   REGION Output Mapping
       // TwoWayActuator
       "Unit1.Em0.HmiInterface".cmStacker1NgBoxClampMoverOpenClose.commands := "ManualOperationControl_U1Em0".twoWayActuator[1].commands;
       "Unit1.Em0.HmiInterface".cmStacker1NgBoxClampLeftOpenClose.commands := "ManualOperationControl_U1Em0".twoWayActuator[2].commands;
       "Unit1.Em0.HmiInterface".cmStacker1NgBoxClampRightOpenClose.commands := "ManualOperationControl_U1Em0".twoWayActuator[3].commands;
       "Unit1.Em0.HmiInterface".cmStacker1NgBoxLoadingUpDown.commands := "ManualOperationControl_U1Em0".twoWayActuator[4].commands;
       "Unit1.Em0.HmiInterface".cmStacker1NgBoxUnitMoverBwdFwd.commands := "ManualOperationControl_U1Em0".twoWayActuator[5].commands;
       "Unit1.Em0.HmiInterface".cmStacker1NgBoxLiftDownUp.commands := "ManualOperationControl_U1Em0".twoWayActuator[6].commands;
       "Unit1.Em0.HmiInterface".cmStacker1NgBoxLockDownUp.commands := "ManualOperationControl_U1Em0".twoWayActuator[7].commands;
   END_REGION
END_REGION

REGION Network 3: Equipment Module 0
   RUNG wire#powerrail
      "CallManualOperationLines_EM"(disableUnit := #disableUnit1, manualOperationEm := "ManualOperationControl_U1Em0".manualOperationEm, manualOperationEmArea := "ManualOperationControl_U1Em0".manualOperationEmArea, manualOperationCms := "ManualOperationControl_U1Em0".manualOperationCms, Axis64Pos := "ManualOperationControl_U1Em0".axis, AxisSoftCam := "ManualOperationControl_U1Em0".softCam, twoWayAcutor := "ManualOperationControl_U1Em0".twoWayActuator, Status := #StatusEm[0].Status, errorID := #errorIDEm[0].errorID)
   END_RUNG
   // the same network as SCL:
   "CallManualOperationLines_EM"(disableUnit := #disableUnit1,
                           manualOperationEm := "ManualOperationControl_U1Em0".manualOperationEm,
                           manualOperationEmArea := "ManualOperationControl_U1Em0".manualOperationEmArea,
                           manualOperationCms := "ManualOperationControl_U1Em0".manualOperationCms,
                           Axis64Pos := "ManualOperationControl_U1Em0".axis,
                           AxisSoftCam := "ManualOperationControl_U1Em0".softCam,
                           twoWayAcutor := "ManualOperationControl_U1Em0".twoWayActuator,
                           Status := #StatusEm[0].Status,
                           errorID := #errorIDEm[0].errorID);
END_REGION

REGION Network 4 (SCL): Equipment Module 1 Cms Mapping
   REGION Input Mapping
       // TwoWayActuator
       "ManualOperationControl_U1Em1".twoWayActuator[1].monitoring := "Unit1.Em1.HmiInterface".cmStacker2NgBoxClampMoverOpenClose.monitoring;
       "ManualOperationControl_U1Em1".twoWayActuator[2].monitoring := "Unit1.Em1.HmiInterface".cmStacker2NgBoxClampLeftOpenClose.monitoring;
       "ManualOperationControl_U1Em1".twoWayActuator[3].monitoring := "Unit1.Em1.HmiInterface".cmStacker2NgBoxClampRightOpenClose.monitoring;
       "ManualOperationControl_U1Em1".twoWayActuator[4].monitoring := "Unit1.Em1.HmiInterface".cmStacker2NgBoxLoadingUpDown.monitoring;
       "ManualOperationControl_U1Em1".twoWayActuator[5].monitoring := "Unit1.Em1.HmiInterface".cmStacker2NgBoxUnitMoverBwdFwd.monitoring;
       "ManualOperationControl_U1Em1".twoWayActuator[6].monitoring := "Unit1.Em1.HmiInterface".cmStacker2NgBoxLiftDownUp.monitoring;
       "ManualOperationControl_U1Em1".twoWayActuator[7].monitoring := "Unit1.Em1.HmiInterface".cmStacker2NgBoxLockDownUp.monitoring;
   END_REGION


   REGION Output Mapping  
       // TwoWayActuator
       "Unit1.Em1.HmiInterface".cmStacker2NgBoxClampMoverOpenClose.commands := "ManualOperationControl_U1Em1".twoWayActuator[1].commands;
       "Unit1.Em1.HmiInterface".cmStacker2NgBoxClampLeftOpenClose.commands := "ManualOperationControl_U1Em1".twoWayActuator[2].commands;
       "Unit1.Em1.HmiInterface".cmStacker2NgBoxClampRightOpenClose.commands := "ManualOperationControl_U1Em1".twoWayActuator[3].commands;
       "Unit1.Em1.HmiInterface".cmStacker2NgBoxLoadingUpDown.commands := "ManualOperationControl_U1Em1".twoWayActuator[4].commands;
       "Unit1.Em1.HmiInterface".cmStacker2NgBoxUnitMoverBwdFwd.commands := "ManualOperationControl_U1Em1".twoWayActuator[5].commands;
       "Unit1.Em1.HmiInterface".cmStacker2NgBoxLiftDownUp.commands := "ManualOperationControl_U1Em1".twoWayActuator[6].commands;
       "Unit1.Em1.HmiInterface".cmStacker2NgBoxLockDownUp.commands := "ManualOperationControl_U1Em1".twoWayActuator[7].commands;
   END_REGION
END_REGION

REGION Network 5: Equipment Module 1
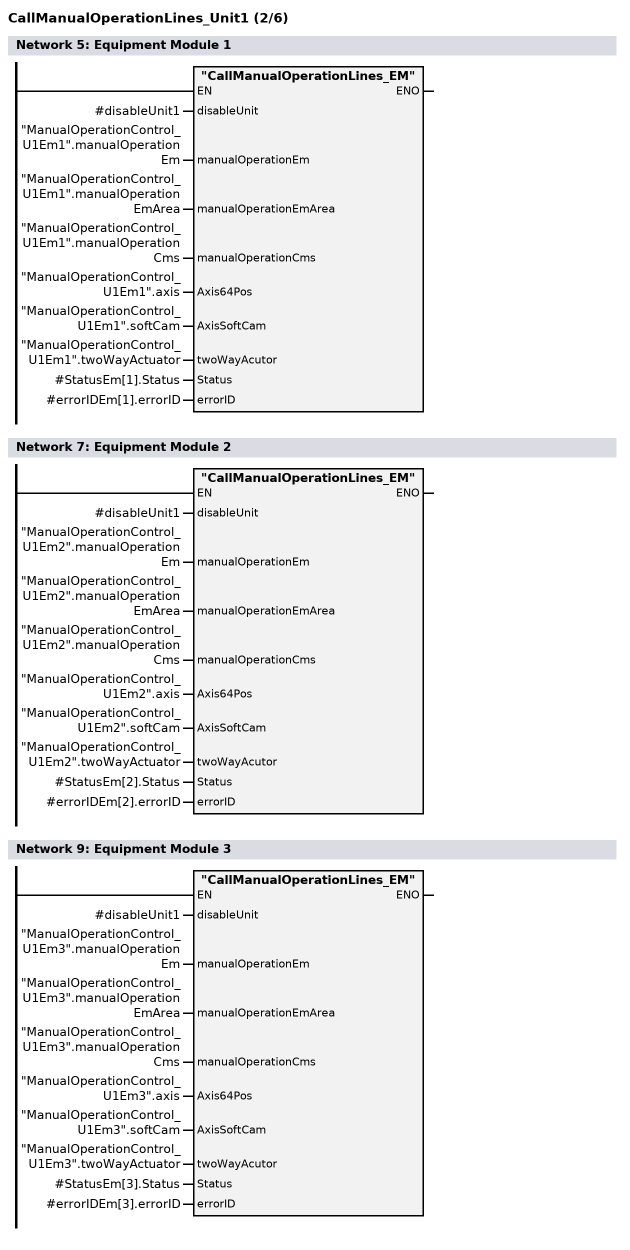
   RUNG wire#powerrail
      "CallManualOperationLines_EM"(disableUnit := #disableUnit1, manualOperationEm := "ManualOperationControl_U1Em1".manualOperationEm, manualOperationEmArea := "ManualOperationControl_U1Em1".manualOperationEmArea, manualOperationCms := "ManualOperationControl_U1Em1".manualOperationCms, Axis64Pos := "ManualOperationControl_U1Em1".axis, AxisSoftCam := "ManualOperationControl_U1Em1".softCam, twoWayAcutor := "ManualOperationControl_U1Em1".twoWayActuator, Status := #StatusEm[1].Status, errorID := #errorIDEm[1].errorID)
   END_RUNG
   // the same network as SCL:
   "CallManualOperationLines_EM"(disableUnit := #disableUnit1,
                           manualOperationEm := "ManualOperationControl_U1Em1".manualOperationEm,
                           manualOperationEmArea := "ManualOperationControl_U1Em1".manualOperationEmArea,
                           manualOperationCms := "ManualOperationControl_U1Em1".manualOperationCms,
                           Axis64Pos := "ManualOperationControl_U1Em1".axis,
                           AxisSoftCam := "ManualOperationControl_U1Em1".softCam,
                           twoWayAcutor := "ManualOperationControl_U1Em1".twoWayActuator,
                           Status := #StatusEm[1].Status,
                           errorID := #errorIDEm[1].errorID);
END_REGION

REGION Network 6 (SCL): Equipment Module 2 Cms Mapping
   REGION Input Mapping
       // Axis
       "ManualOperationControl_U1Em2".axis[1].monitoring := "Unit1.Em2.HmiInterface".cmJROutPnPLeftAxisX.monitoring;
       "ManualOperationControl_U1Em2".axis[2].monitoring := "Unit1.Em2.HmiInterface".cmJROutPnPLeftAxisZ.monitoring;
       "ManualOperationControl_U1Em2".axis[3].monitoring := "Unit1.Em2.HmiInterface".cmJROutPnPRightAxisX.monitoring;
       "ManualOperationControl_U1Em2".axis[4].monitoring := "Unit1.Em2.HmiInterface".cmJROutPnPRightAxisZ.monitoring;

       // SoftCam
       "ManualOperationControl_U1Em2".softCam[1] := "Unit1.Em2.HmiInterface".cm.softcam.jrOutPnPLeftAxisX;
       "ManualOperationControl_U1Em2".softCam[2] := "Unit1.Em2.HmiInterface".cm.softcam.jrOutPnPLeftAxisZ;
       "ManualOperationControl_U1Em2".softCam[3] := "Unit1.Em2.HmiInterface".cm.softcam.jrOutPnPRightAxisX;
       "ManualOperationControl_U1Em2".softCam[4] := "Unit1.Em2.HmiInterface".cm.softcam.jrOutPnPRightAxisZ;

       // TwoWayActuator
       "ManualOperationControl_U1Em2".twoWayActuator[1].monitoring := "Unit1.Em2.HmiInterface".cmJROutPnPLeftClampOpenClose.monitoring;
       "ManualOperationControl_U1Em2".twoWayActuator[2].monitoring := "Unit1.Em2.HmiInterface".cmJROutPnPRightClampOpenClose.monitoring;
   END_REGION


   REGION Output Mapping
       // Axis
       "Unit1.Em2.HmiInterface".cmJROutPnPLeftAxisX.commands.jogForward := "ManualOperationControl_U1Em2".axis[1].commands.jogForward;
       "Unit1.Em2.HmiInterface".cmJROutPnPLeftAxisX.commands.jogBackward := "ManualOperationControl_U1Em2".axis[1].commands.jogBackward;
       "Unit1.Em2.HmiInterface".cmJROutPnPLeftAxisZ.commands.jogForward := "ManualOperationControl_U1Em2".axis[2].commands.jogForward;
       "Unit1.Em2.HmiInterface".cmJROutPnPLeftAxisZ.commands.jogBackward := "ManualOperationControl_U1Em2".axis[2].commands.jogBackward;
       "Unit1.Em2.HmiInterface".cmJROutPnPRightAxisX.commands.jogForward := "ManualOperationControl_U1Em2".axis[3].commands.jogForward;
       "Unit1.Em2.HmiInterface".cmJROutPnPRightAxisX.commands.jogBackward := "ManualOperationControl_U1Em2".axis[3].commands.jogBackward;
       "Unit1.Em2.HmiInterface".cmJROutPnPRightAxisZ.commands.jogForward := "ManualOperationControl_U1Em2".axis[4].commands.jogForward;
       "Unit1.Em2.HmiInterface".cmJROutPnPRightAxisZ.commands.jogBackward := "ManualOperationControl_U1Em2".axis[4].commands.jogBackward;

       // TwoWayActuator
       "Unit1.Em2.HmiInterface".cmJROutPnPLeftClampOpenClose.commands := "ManualOperationControl_U1Em2".twoWayActuator[1].commands;
       "Unit1.Em2.HmiInterface".cmJROutPnPRightClampOpenClose.commands := "ManualOperationControl_U1Em2".twoWayActuator[2].commands;
   END_REGION
END_REGION

REGION Network 7: Equipment Module 2
   RUNG wire#powerrail
      "CallManualOperationLines_EM"(disableUnit := #disableUnit1, manualOperationEm := "ManualOperationControl_U1Em2".manualOperationEm, manualOperationEmArea := "ManualOperationControl_U1Em2".manualOperationEmArea, manualOperationCms := "ManualOperationControl_U1Em2".manualOperationCms, Axis64Pos := "ManualOperationControl_U1Em2".axis, AxisSoftCam := "ManualOperationControl_U1Em2".softCam, twoWayAcutor := "ManualOperationControl_U1Em2".twoWayActuator, Status := #StatusEm[2].Status, errorID := #errorIDEm[2].errorID)
   END_RUNG
   // the same network as SCL:
   "CallManualOperationLines_EM"(disableUnit := #disableUnit1,
                           manualOperationEm := "ManualOperationControl_U1Em2".manualOperationEm,
                           manualOperationEmArea := "ManualOperationControl_U1Em2".manualOperationEmArea,
                           manualOperationCms := "ManualOperationControl_U1Em2".manualOperationCms,
                           Axis64Pos := "ManualOperationControl_U1Em2".axis,
                           AxisSoftCam := "ManualOperationControl_U1Em2".softCam,
                           twoWayAcutor := "ManualOperationControl_U1Em2".twoWayActuator,
                           Status := #StatusEm[2].Status,
                           errorID := #errorIDEm[2].errorID);
END_REGION

REGION Network 8 (SCL): Equipment Module 3 Cms Mapping
   REGION Input Mapping
        // Axis
       "ManualOperationControl_U1Em3".axis[1].monitoring := "Unit1.Em3.HmiInterface".cmTopTapeAxisX.monitoring;
       "ManualOperationControl_U1Em3".axis[2].monitoring := "Unit1.Em3.HmiInterface".cmTopTapeAxisY.monitoring;

       // SoftCam
       "ManualOperationControl_U1Em3".softCam[1] := "Unit1.Em3.HmiInterface".cm.softcam.topTapeAxisX;
       "ManualOperationControl_U1Em3".softCam[2] := "Unit1.Em3.HmiInterface".cm.softcam.topTapeAxisY;

       // TwoWayActuator
       "ManualOperationControl_U1Em3".twoWayActuator[1].monitoring := "Unit1.Em3.HmiInterface".cmTopTapeCutterUpDown.monitoring;
       "ManualOperationControl_U1Em3".twoWayActuator[2].monitoring := "Unit1.Em3.HmiInterface".cmTopTapeCutterClampUpDown.monitoring;
       "ManualOperationControl_U1Em3".twoWayActuator[3].monitoring := "Unit1.Em3.HmiInterface".cmTopTapeLoadingClampOpenClose.monitoring;
       "ManualOperationControl_U1Em3".twoWayActuator[4].monitoring := "Unit1.Em3.HmiInterface".cmTopTapeTensionBwdFwd.monitoring;
       "ManualOperationControl_U1Em3".twoWayActuator[5].monitoring := "Unit1.Em3.HmiInterface".cmTopTapeLoadingBwdFwd.monitoring;
       "ManualOperationControl_U1Em3".twoWayActuator[6].monitoring := "Unit1.Em3.HmiInterface".cmTopTapeClampTopLeftUpDown.monitoring;
       "ManualOperationControl_U1Em3".twoWayActuator[7].monitoring := "Unit1.Em3.HmiInterface".cmTopTapeClampTopCenterUpDown.monitoring;
       "ManualOperationControl_U1Em3".twoWayActuator[8].monitoring := "Unit1.Em3.HmiInterface".cmTopTapeClampTopRightUpDown.monitoring;
       "ManualOperationControl_U1Em3".twoWayActuator[9].monitoring := "Unit1.Em3.HmiInterface".cmTopTapeClampBtmDownUp.monitoring;
       "ManualOperationControl_U1Em3".twoWayActuator[10].monitoring := "Unit1.Em3.HmiInterface".cmTopTapeAttachmentUpDown.monitoring;
       "ManualOperationControl_U1Em3".twoWayActuator[11].monitoring := "Unit1.Em3.HmiInterface".cmTopTapeAttachmentVaccumOffOn.monitoring;

   END_REGION


   REGION Output Mapping
       // Axis
       "Unit1.Em3.HmiInterface".cmTopTapeAxisX.commands.jogForward := "ManualOperationControl_U1Em3".axis[1].commands.jogForward;
       "Unit1.Em3.HmiInterface".cmTopTapeAxisX.commands.jogBackward := "ManualOperationControl_U1Em3".axis[1].commands.jogBackward;
       "Unit1.Em3.HmiInterface".cmTopTapeAxisY.commands.jogForward := "ManualOperationControl_U1Em3".axis[2].commands.jogForward;
       "Unit1.Em3.HmiInterface".cmTopTapeAxisY.commands.jogBackward := "ManualOperationControl_U1Em3".axis[2].commands.jogBackward;

       // TwoWayActuator
       "Unit1.Em3.HmiInterface".cmTopTapeCutterUpDown.commands := "ManualOperationControl_U1Em3".twoWayActuator[1].commands;
       "Unit1.Em3.HmiInterface".cmTopTapeCutterClampUpDown.commands := "ManualOperationControl_U1Em3".twoWayActuator[2].commands;
       "Unit1.Em3.HmiInterface".cmTopTapeLoadingClampOpenClose.commands := "ManualOperationControl_U1Em3".twoWayActuator[3].commands;
       "Unit1.Em3.HmiInterface".cmTopTapeTensionBwdFwd.commands := "ManualOperationControl_U1Em3".twoWayActuator[4].commands;
       "Unit1.Em3.HmiInterface".cmTopTapeLoadingBwdFwd.commands := "ManualOperationControl_U1Em3".twoWayActuator[5].commands;
       "Unit1.Em3.HmiInterface".cmTopTapeClampTopLeftUpDown.commands := "ManualOperationControl_U1Em3".twoWayActuator[6].commands;
       "Unit1.Em3.HmiInterface".cmTopTapeClampTopCenterUpDown.commands := "ManualOperationControl_U1Em3".twoWayActuator[7].commands;
       "Unit1.Em3.HmiInterface".cmTopTapeClampTopRightUpDown.commands := "ManualOperationControl_U1Em3".twoWayActuator[8].commands;
       "Unit1.Em3.HmiInterface".cmTopTapeClampBtmDownUp.commands := "ManualOperationControl_U1Em3".twoWayActuator[9].commands;
       "Unit1.Em3.HmiInterface".cmTopTapeAttachmentUpDown.commands := "ManualOperationControl_U1Em3".twoWayActuator[10].commands;
       "Unit1.Em3.HmiInterface".cmTopTapeAttachmentVaccumOffOn.commands := "ManualOperationControl_U1Em3".twoWayActuator[11].commands;

   END_REGION
END_REGION

REGION Network 9: Equipment Module 3
   RUNG wire#powerrail
      "CallManualOperationLines_EM"(disableUnit := #disableUnit1, manualOperationEm := "ManualOperationControl_U1Em3".manualOperationEm, manualOperationEmArea := "ManualOperationControl_U1Em3".manualOperationEmArea, manualOperationCms := "ManualOperationControl_U1Em3".manualOperationCms, Axis64Pos := "ManualOperationControl_U1Em3".axis, AxisSoftCam := "ManualOperationControl_U1Em3".softCam, twoWayAcutor := "ManualOperationControl_U1Em3".twoWayActuator, Status := #StatusEm[3].Status, errorID := #errorIDEm[3].errorID)
   END_RUNG
   // the same network as SCL:
   "CallManualOperationLines_EM"(disableUnit := #disableUnit1,
                           manualOperationEm := "ManualOperationControl_U1Em3".manualOperationEm,
                           manualOperationEmArea := "ManualOperationControl_U1Em3".manualOperationEmArea,
                           manualOperationCms := "ManualOperationControl_U1Em3".manualOperationCms,
                           Axis64Pos := "ManualOperationControl_U1Em3".axis,
                           AxisSoftCam := "ManualOperationControl_U1Em3".softCam,
                           twoWayAcutor := "ManualOperationControl_U1Em3".twoWayActuator,
                           Status := #StatusEm[3].Status,
                           errorID := #errorIDEm[3].errorID);
END_REGION

REGION Network 10 (SCL): Equipment Module 4 Cms Mapping
   REGION Input Mapping
       // Axis
       "ManualOperationControl_U1Em4".axis[1].monitoring := "Unit1.Em4.HmiInterface".cmSideTapeFixStageAxisX.monitoring;
       "ManualOperationControl_U1Em4".axis[2].monitoring := "Unit1.Em4.HmiInterface".cmSideTapeFixStageAxisC.monitoring;
       "ManualOperationControl_U1Em4".axis[3].monitoring := "Unit1.Em4.HmiInterface".cmSideTapeAttachmentAxisX.monitoring;
       "ManualOperationControl_U1Em4".axis[4].monitoring := "Unit1.Em4.HmiInterface".cmSideTapeAttachmentAxisY.monitoring;

       // SoftCam
       "ManualOperationControl_U1Em4".softCam[1] := "Unit1.Em4.HmiInterface".cm.softcam.sideTapeFixStageAxisX;
       "ManualOperationControl_U1Em4".softCam[2] := "Unit1.Em4.HmiInterface".cm.softcam.sideTapeFixStageAxisC;
       "ManualOperationControl_U1Em4".softCam[3] := "Unit1.Em4.HmiInterface".cm.softcam.sideTapeAttachmentAxisX;
       "ManualOperationControl_U1Em4".softCam[4] := "Unit1.Em4.HmiInterface".cm.softcam.sideTapeAttachmentAxisY;

       // TwoWayActuator
       "ManualOperationControl_U1Em4".twoWayActuator[1].monitoring := "Unit1.Em4.HmiInterface".cmSideTapeCutterBwdFwd.monitoring;
       "ManualOperationControl_U1Em4".twoWayActuator[2].monitoring := "Unit1.Em4.HmiInterface".cmSideTapeCutterClampBwdFwd.monitoring;
       "ManualOperationControl_U1Em4".twoWayActuator[3].monitoring := "Unit1.Em4.HmiInterface".cmSideTapeLoadingClampOpenClose.monitoring;
       "ManualOperationControl_U1Em4".twoWayActuator[4].monitoring := "Unit1.Em4.HmiInterface".cmSideTapeLoadingDownUp.monitoring;
       "ManualOperationControl_U1Em4".twoWayActuator[5].monitoring := "Unit1.Em4.HmiInterface".cmSideTapeTensionBwdFwd.monitoring;
       "ManualOperationControl_U1Em4".twoWayActuator[6].monitoring := "Unit1.Em4.HmiInterface".cmSideTapeAttachmentLeftBwdFwd.monitoring;
       "ManualOperationControl_U1Em4".twoWayActuator[7].monitoring := "Unit1.Em4.HmiInterface".cmSideTapeAttachmentRightBwdFwd.monitoring;
       "ManualOperationControl_U1Em4".twoWayActuator[8].monitoring := "Unit1.Em4.HmiInterface".cmSideTapeAttachmentBtmBwdFwd.monitoring;
       "ManualOperationControl_U1Em4".twoWayActuator[9].monitoring := "Unit1.Em4.HmiInterface".cmSideTapeFixStageClampOpenClose.monitoring;
       "ManualOperationControl_U1Em4".twoWayActuator[10].monitoring := "Unit1.Em4.HmiInterface".cmSideTapeAttachment1TopVaccumOffOn.monitoring;
       "ManualOperationControl_U1Em4".twoWayActuator[11].monitoring := "Unit1.Em4.HmiInterface".cmSideTapeAttachment1BtmVaccumOffOn.monitoring;
       "ManualOperationControl_U1Em4".twoWayActuator[12].monitoring := "Unit1.Em4.HmiInterface".cmSideTapeAttachment2TopVaccumOffOn.monitoring;
       "ManualOperationControl_U1Em4".twoWayActuator[13].monitoring := "Unit1.Em4.HmiInterface".cmSideTapeAttachment2BtmVaccumOffOn.monitoring;

   END_REGION


   REGION Output Mapping
       // Axis
       "Unit1.Em4.HmiInterface".cmSideTapeFixStageAxisX.commands.jogForward := "ManualOperationControl_U1Em4".axis[1].commands.jogForward;
       "Unit1.Em4.HmiInterface".cmSideTapeFixStageAxisX.commands.jogBackward := "ManualOperationControl_U1Em4".axis[1].commands.jogBackward;
       "Unit1.Em4.HmiInterface".cmSideTapeFixStageAxisC.commands.jogForward := "ManualOperationControl_U1Em4".axis[2].commands.jogForward;
       "Unit1.Em4.HmiInterface".cmSideTapeFixStageAxisC.commands.jogBackward := "ManualOperationControl_U1Em4".axis[2].commands.jogBackward;
       "Unit1.Em4.HmiInterface".cmSideTapeAttachmentAxisX.commands.jogForward := "ManualOperationControl_U1Em4".axis[3].commands.jogForward;
       "Unit1.Em4.HmiInterface".cmSideTapeAttachmentAxisX.commands.jogBackward := "ManualOperationControl_U1Em4".axis[3].commands.jogBackward;
       "Unit1.Em4.HmiInterface".cmSideTapeAttachmentAxisY.commands.jogForward := "ManualOperationControl_U1Em4".axis[4].commands.jogForward;
       "Unit1.Em4.HmiInterface".cmSideTapeAttachmentAxisY.commands.jogBackward := "ManualOperationControl_U1Em4".axis[4].commands.jogBackward;

       // TwoWayActuator
       "Unit1.Em4.HmiInterface".cmSideTapeCutterBwdFwd.commands := "ManualOperationControl_U1Em4".twoWayActuator[1].commands;
       "Unit1.Em4.HmiInterface".cmSideTapeCutterClampBwdFwd.commands := "ManualOperationControl_U1Em4".twoWayActuator[2].commands;
       "Unit1.Em4.HmiInterface".cmSideTapeLoadingClampOpenClose.commands := "ManualOperationControl_U1Em4".twoWayActuator[3].commands;
       "Unit1.Em4.HmiInterface".cmSideTapeLoadingDownUp.commands:= "ManualOperationControl_U1Em4".twoWayActuator[4].commands;
       "Unit1.Em4.HmiInterface".cmSideTapeTensionBwdFwd.commands := "ManualOperationControl_U1Em4".twoWayActuator[5].commands;
       "Unit1.Em4.HmiInterface".cmSideTapeAttachmentLeftBwdFwd.commands := "ManualOperationControl_U1Em4".twoWayActuator[6].commands;
       "Unit1.Em4.HmiInterface".cmSideTapeAttachmentRightBwdFwd.commands := "ManualOperationControl_U1Em4".twoWayActuator[7].commands;
       "Unit1.Em4.HmiInterface".cmSideTapeAttachmentBtmBwdFwd.commands := "ManualOperationControl_U1Em4".twoWayActuator[8].commands;
       "Unit1.Em4.HmiInterface".cmSideTapeFixStageClampOpenClose.commands := "ManualOperationControl_U1Em4".twoWayActuator[9].commands;
       "Unit1.Em4.HmiInterface".cmSideTapeAttachment1TopVaccumOffOn.commands := "ManualOperationControl_U1Em4".twoWayActuator[10].commands;
       "Unit1.Em4.HmiInterface".cmSideTapeAttachment1BtmVaccumOffOn.commands := "ManualOperationControl_U1Em4".twoWayActuator[11].commands;
       "Unit1.Em4.HmiInterface".cmSideTapeAttachment2TopVaccumOffOn.commands := "ManualOperationControl_U1Em4".twoWayActuator[12].commands;
       "Unit1.Em4.HmiInterface".cmSideTapeAttachment2BtmVaccumOffOn.commands := "ManualOperationControl_U1Em4".twoWayActuator[13].commands;

   END_REGION
END_REGION

REGION Network 11: Equipment Module 4
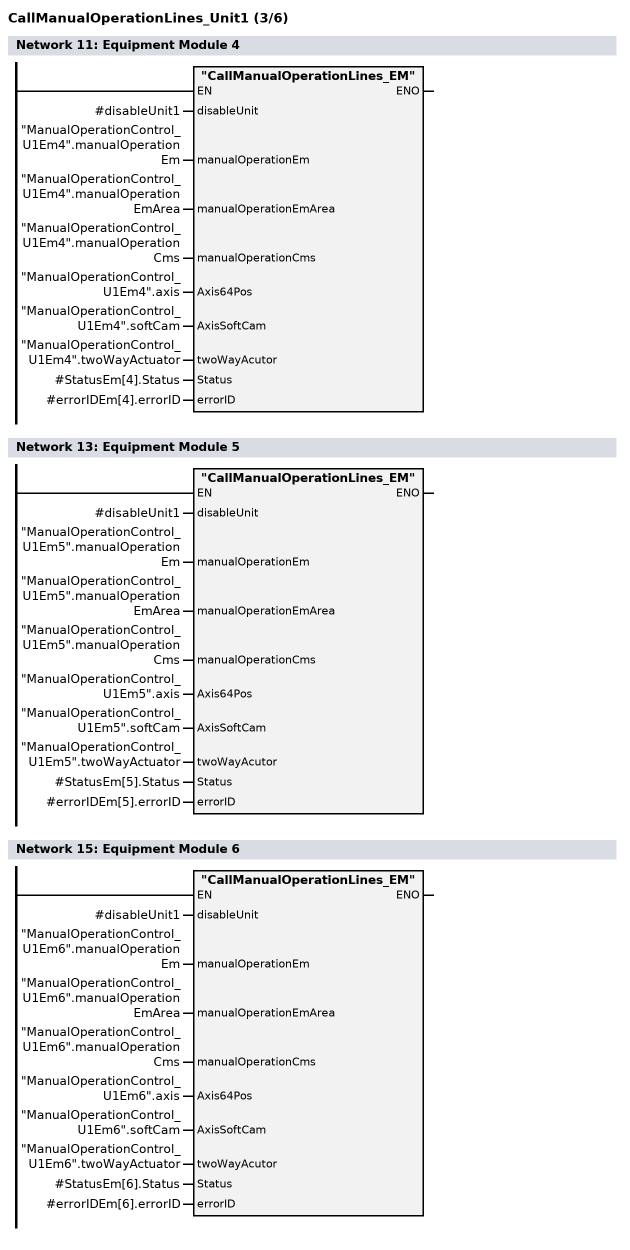
   RUNG wire#powerrail
      "CallManualOperationLines_EM"(disableUnit := #disableUnit1, manualOperationEm := "ManualOperationControl_U1Em4".manualOperationEm, manualOperationEmArea := "ManualOperationControl_U1Em4".manualOperationEmArea, manualOperationCms := "ManualOperationControl_U1Em4".manualOperationCms, Axis64Pos := "ManualOperationControl_U1Em4".axis, AxisSoftCam := "ManualOperationControl_U1Em4".softCam, twoWayAcutor := "ManualOperationControl_U1Em4".twoWayActuator, Status := #StatusEm[4].Status, errorID := #errorIDEm[4].errorID)
   END_RUNG
   // the same network as SCL:
   "CallManualOperationLines_EM"(disableUnit := #disableUnit1,
                           manualOperationEm := "ManualOperationControl_U1Em4".manualOperationEm,
                           manualOperationEmArea := "ManualOperationControl_U1Em4".manualOperationEmArea,
                           manualOperationCms := "ManualOperationControl_U1Em4".manualOperationCms,
                           Axis64Pos := "ManualOperationControl_U1Em4".axis,
                           AxisSoftCam := "ManualOperationControl_U1Em4".softCam,
                           twoWayAcutor := "ManualOperationControl_U1Em4".twoWayActuator,
                           Status := #StatusEm[4].Status,
                           errorID := #errorIDEm[4].errorID);
END_REGION

REGION Network 12 (SCL): Equipment Module 5 Cms Mapping
   REGION Input Mapping
        // Axis
       "ManualOperationControl_U1Em5".axis[1].monitoring := "Unit1.Em5.HmiInterface".cmTransferPnPLeftAxisX.monitoring;
       "ManualOperationControl_U1Em5".axis[2].monitoring := "Unit1.Em5.HmiInterface".cmTransferPnPLeftAxisY.monitoring;
       "ManualOperationControl_U1Em5".axis[3].monitoring := "Unit1.Em5.HmiInterface".cmTransferPnPLeftAxisZ.monitoring;
       "ManualOperationControl_U1Em5".axis[4].monitoring := "Unit1.Em5.HmiInterface".cmTransferPnPRightAxisX.monitoring;
       "ManualOperationControl_U1Em5".axis[5].monitoring := "Unit1.Em5.HmiInterface".cmTransferPnPRightAxisY.monitoring;
       "ManualOperationControl_U1Em5".axis[6].monitoring := "Unit1.Em5.HmiInterface".cmTransferPnPRightAxisZ.monitoring;

       // SoftCam
       "ManualOperationControl_U1Em5".softCam[1] := "Unit1.Em5.HmiInterface".cm.softcam.transferPnPLeftAxisX;
       "ManualOperationControl_U1Em5".softCam[2] := "Unit1.Em5.HmiInterface".cm.softcam.transferPnPLeftAxisY;
       "ManualOperationControl_U1Em5".softCam[3] := "Unit1.Em5.HmiInterface".cm.softcam.transferPnPLeftAxisZ;
       "ManualOperationControl_U1Em5".softCam[4] := "Unit1.Em5.HmiInterface".cm.softcam.transferPnPRightAxisX;
       "ManualOperationControl_U1Em5".softCam[5] := "Unit1.Em5.HmiInterface".cm.softcam.transferPnPRightAxisY;
       "ManualOperationControl_U1Em5".softCam[6] := "Unit1.Em5.HmiInterface".cm.softcam.transferPnPRightAxisZ;

       // TwoWayActuator
       "ManualOperationControl_U1Em5".twoWayActuator[1].monitoring := "Unit1.Em5.HmiInterface".cmTransferPnPLeftClampOpenClose.monitoring;
       "ManualOperationControl_U1Em5".twoWayActuator[2].monitoring := "Unit1.Em5.HmiInterface".cmTransferPnPRightClampOpenClose.monitoring;
   END_REGION


   REGION Output Mapping
       // Axis
       "Unit1.Em5.HmiInterface".cmTransferPnPLeftAxisX.commands.jogForward := "ManualOperationControl_U1Em5".axis[1].commands.jogForward;
       "Unit1.Em5.HmiInterface".cmTransferPnPLeftAxisX.commands.jogBackward := "ManualOperationControl_U1Em5".axis[1].commands.jogBackward;
       "Unit1.Em5.HmiInterface".cmTransferPnPLeftAxisY.commands.jogForward := "ManualOperationControl_U1Em5".axis[2].commands.jogForward;
       "Unit1.Em5.HmiInterface".cmTransferPnPLeftAxisY.commands.jogBackward := "ManualOperationControl_U1Em5".axis[2].commands.jogBackward;
       "Unit1.Em5.HmiInterface".cmTransferPnPLeftAxisZ.commands.jogForward := "ManualOperationControl_U1Em5".axis[3].commands.jogForward;
       "Unit1.Em5.HmiInterface".cmTransferPnPLeftAxisZ.commands.jogBackward := "ManualOperationControl_U1Em5".axis[3].commands.jogBackward;
       "Unit1.Em5.HmiInterface".cmTransferPnPRightAxisX.commands.jogForward := "ManualOperationControl_U1Em5".axis[4].commands.jogForward;
       "Unit1.Em5.HmiInterface".cmTransferPnPRightAxisX.commands.jogBackward := "ManualOperationControl_U1Em5".axis[4].commands.jogBackward;
       "Unit1.Em5.HmiInterface".cmTransferPnPRightAxisY.commands.jogForward := "ManualOperationControl_U1Em5".axis[5].commands.jogForward;
       "Unit1.Em5.HmiInterface".cmTransferPnPRightAxisY.commands.jogBackward := "ManualOperationControl_U1Em5".axis[5].commands.jogBackward;
       "Unit1.Em5.HmiInterface".cmTransferPnPRightAxisZ.commands.jogForward := "ManualOperationControl_U1Em5".axis[6].commands.jogForward;
       "Unit1.Em5.HmiInterface".cmTransferPnPRightAxisZ.commands.jogBackward := "ManualOperationControl_U1Em5".axis[6].commands.jogBackward;

       // TwoWayActuator
       "Unit1.Em5.HmiInterface".cmTransferPnPLeftClampOpenClose.commands := "ManualOperationControl_U1Em5".twoWayActuator[1].commands;
       "Unit1.Em5.HmiInterface".cmTransferPnPRightClampOpenClose.commands := "ManualOperationControl_U1Em5".twoWayActuator[2].commands;
   END_REGION
END_REGION

REGION Network 13: Equipment Module 5
   RUNG wire#powerrail
      "CallManualOperationLines_EM"(disableUnit := #disableUnit1, manualOperationEm := "ManualOperationControl_U1Em5".manualOperationEm, manualOperationEmArea := "ManualOperationControl_U1Em5".manualOperationEmArea, manualOperationCms := "ManualOperationControl_U1Em5".manualOperationCms, Axis64Pos := "ManualOperationControl_U1Em5".axis, AxisSoftCam := "ManualOperationControl_U1Em5".softCam, twoWayAcutor := "ManualOperationControl_U1Em5".twoWayActuator, Status := #StatusEm[5].Status, errorID := #errorIDEm[5].errorID)
   END_RUNG
   // the same network as SCL:
   "CallManualOperationLines_EM"(disableUnit := #disableUnit1,
                           manualOperationEm := "ManualOperationControl_U1Em5".manualOperationEm,
                           manualOperationEmArea := "ManualOperationControl_U1Em5".manualOperationEmArea,
                           manualOperationCms := "ManualOperationControl_U1Em5".manualOperationCms,
                           Axis64Pos := "ManualOperationControl_U1Em5".axis,
                           AxisSoftCam := "ManualOperationControl_U1Em5".softCam,
                           twoWayAcutor := "ManualOperationControl_U1Em5".twoWayActuator,
                           Status := #StatusEm[5].Status,
                           errorID := #errorIDEm[5].errorID);
END_REGION

REGION Network 14 (SCL): Equipment Module 6 Cms Mapping
   REGION Input Mapping  
       // TwoWayActuator
       "ManualOperationControl_U1Em6".twoWayActuator[3].monitoring := "Unit1.Em6.HmiInterface".cmHotpressLeftStageLiftFrontUpDown.monitoring;
       "ManualOperationControl_U1Em6".twoWayActuator[4].monitoring := "Unit1.Em6.HmiInterface".cmHotpressLeftStageLiftRearUpDown.monitoring;
   END_REGION


   REGION Output Mapping
       // TwoWayActuator
       "Unit1.Em6.HmiInterface".cmHotpressLeftStageLiftFrontUpDown.commands := "ManualOperationControl_U1Em6".twoWayActuator[3].commands;
       "Unit1.Em6.HmiInterface".cmHotpressLeftStageLiftRearUpDown.commands := "ManualOperationControl_U1Em6".twoWayActuator[4].commands;
   END_REGION
END_REGION

REGION Network 15: Equipment Module 6
   RUNG wire#powerrail
      "CallManualOperationLines_EM"(disableUnit := #disableUnit1, manualOperationEm := "ManualOperationControl_U1Em6".manualOperationEm, manualOperationEmArea := "ManualOperationControl_U1Em6".manualOperationEmArea, manualOperationCms := "ManualOperationControl_U1Em6".manualOperationCms, Axis64Pos := "ManualOperationControl_U1Em6".axis, AxisSoftCam := "ManualOperationControl_U1Em6".softCam, twoWayAcutor := "ManualOperationControl_U1Em6".twoWayActuator, Status := #StatusEm[6].Status, errorID := #errorIDEm[6].errorID)
   END_RUNG
   // the same network as SCL:
   "CallManualOperationLines_EM"(disableUnit := #disableUnit1,
                           manualOperationEm := "ManualOperationControl_U1Em6".manualOperationEm,
                           manualOperationEmArea := "ManualOperationControl_U1Em6".manualOperationEmArea,
                           manualOperationCms := "ManualOperationControl_U1Em6".manualOperationCms,
                           Axis64Pos := "ManualOperationControl_U1Em6".axis,
                           AxisSoftCam := "ManualOperationControl_U1Em6".softCam,
                           twoWayAcutor := "ManualOperationControl_U1Em6".twoWayActuator,
                           Status := #StatusEm[6].Status,
                           errorID := #errorIDEm[6].errorID);
END_REGION

REGION Network 16 (SCL): Equipment Module 7 Cms Mapping
   REGION Input Mapping  
       // TwoWayActuator
       "ManualOperationControl_U1Em7".twoWayActuator[3].monitoring := "Unit1.Em7.HmiInterface".cmHotPressRightStageLiftFrontUpDown.monitoring;
       "ManualOperationControl_U1Em7".twoWayActuator[4].monitoring := "Unit1.Em7.HmiInterface".cmHotPressRightStageLiftRearUpDown.monitoring;
   END_REGION


   REGION Output Mapping
       // TwoWayActuator
       "Unit1.Em7.HmiInterface".cmHotPressRightStageLiftFrontUpDown.commands := "ManualOperationControl_U1Em7".twoWayActuator[3].commands;
       "Unit1.Em7.HmiInterface".cmHotPressRightStageLiftRearUpDown.commands := "ManualOperationControl_U1Em7".twoWayActuator[4].commands;
   END_REGION
END_REGION

REGION Network 17: Equipment Module 7
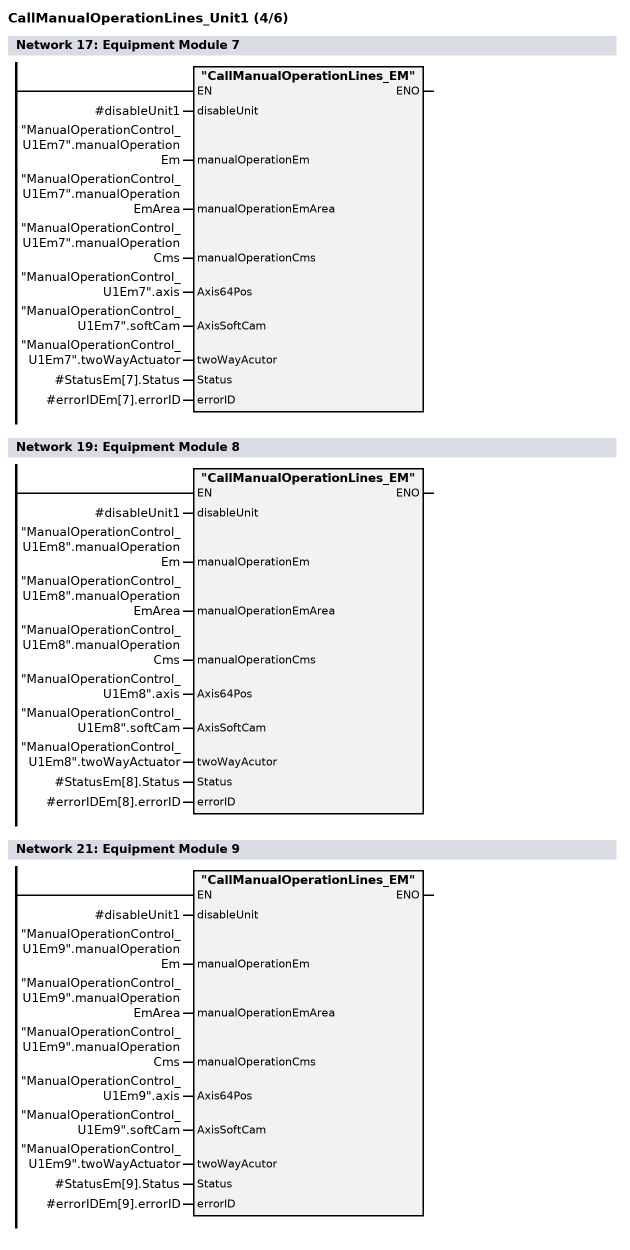
   RUNG wire#powerrail
      "CallManualOperationLines_EM"(disableUnit := #disableUnit1, manualOperationEm := "ManualOperationControl_U1Em7".manualOperationEm, manualOperationEmArea := "ManualOperationControl_U1Em7".manualOperationEmArea, manualOperationCms := "ManualOperationControl_U1Em7".manualOperationCms, Axis64Pos := "ManualOperationControl_U1Em7".axis, AxisSoftCam := "ManualOperationControl_U1Em7".softCam, twoWayAcutor := "ManualOperationControl_U1Em7".twoWayActuator, Status := #StatusEm[7].Status, errorID := #errorIDEm[7].errorID)
   END_RUNG
   // the same network as SCL:
   "CallManualOperationLines_EM"(disableUnit := #disableUnit1,
                           manualOperationEm := "ManualOperationControl_U1Em7".manualOperationEm,
                           manualOperationEmArea := "ManualOperationControl_U1Em7".manualOperationEmArea,
                           manualOperationCms := "ManualOperationControl_U1Em7".manualOperationCms,
                           Axis64Pos := "ManualOperationControl_U1Em7".axis,
                           AxisSoftCam := "ManualOperationControl_U1Em7".softCam,
                           twoWayAcutor := "ManualOperationControl_U1Em7".twoWayActuator,
                           Status := #StatusEm[7].Status,
                           errorID := #errorIDEm[7].errorID);
END_REGION

REGION Network 18 (SCL): Equipment Module 8 Cms Mapping
   REGION Input Mapping
        // Axis
       "ManualOperationControl_U1Em8".axis[1].monitoring := "Unit1.Em8.HmiInterface".cmThicknessAxisZ.monitoring;

       // SoftCam
       "ManualOperationControl_U1Em8".softCam[1] := "Unit1.Em8.HmiInterface".cm.softcam.thicknessAxisZ;

       // TwoWayActuator
       "ManualOperationControl_U1Em8".twoWayActuator[1].monitoring := "Unit1.Em8.HmiInterface".cmHipotTabContactorBwdFwd.monitoring;
       "ManualOperationControl_U1Em8".twoWayActuator[2].monitoring := "Unit1.Em8.HmiInterface".cmHipotTabContactorLeftOpenClose.monitoring;
       "ManualOperationControl_U1Em8".twoWayActuator[3].monitoring := "Unit1.Em8.HmiInterface".cmHipotTabContactorRightOpenClose.monitoring;
       "ManualOperationControl_U1Em8".twoWayActuator[6].monitoring := "Unit1.Em8.HmiInterface".cmHipotThicknessStageLiftFrontUpDown.monitoring;
       "ManualOperationControl_U1Em8".twoWayActuator[7].monitoring := "Unit1.Em8.HmiInterface".cmHipotThicknessStageLiftRearUpDown.monitoring;
   END_REGION


   REGION Output Mapping
       // Axis
       "Unit1.Em8.HmiInterface".cmThicknessAxisZ.commands.jogForward := "ManualOperationControl_U1Em8".axis[1].commands.jogForward;
       "Unit1.Em8.HmiInterface".cmThicknessAxisZ.commands.jogBackward := "ManualOperationControl_U1Em8".axis[1].commands.jogBackward;

       // TwoWayActuator
       "Unit1.Em8.HmiInterface".cmHipotTabContactorBwdFwd.commands := "ManualOperationControl_U1Em8".twoWayActuator[1].commands;
       "Unit1.Em8.HmiInterface".cmHipotTabContactorLeftOpenClose.commands := "ManualOperationControl_U1Em8".twoWayActuator[2].commands;
       "Unit1.Em8.HmiInterface".cmHipotTabContactorRightOpenClose.commands := "ManualOperationControl_U1Em8".twoWayActuator[3].commands;
       "Unit1.Em8.HmiInterface".cmHipotThicknessStageLiftFrontUpDown.commands := "ManualOperationControl_U1Em8".twoWayActuator[6].commands;
       "Unit1.Em8.HmiInterface".cmHipotThicknessStageLiftRearUpDown.commands := "ManualOperationControl_U1Em8".twoWayActuator[7].commands;
   END_REGION
END_REGION

REGION Network 19: Equipment Module 8
   RUNG wire#powerrail
      "CallManualOperationLines_EM"(disableUnit := #disableUnit1, manualOperationEm := "ManualOperationControl_U1Em8".manualOperationEm, manualOperationEmArea := "ManualOperationControl_U1Em8".manualOperationEmArea, manualOperationCms := "ManualOperationControl_U1Em8".manualOperationCms, Axis64Pos := "ManualOperationControl_U1Em8".axis, AxisSoftCam := "ManualOperationControl_U1Em8".softCam, twoWayAcutor := "ManualOperationControl_U1Em8".twoWayActuator, Status := #StatusEm[8].Status, errorID := #errorIDEm[8].errorID)
   END_RUNG
   // the same network as SCL:
   "CallManualOperationLines_EM"(disableUnit := #disableUnit1,
                           manualOperationEm := "ManualOperationControl_U1Em8".manualOperationEm,
                           manualOperationEmArea := "ManualOperationControl_U1Em8".manualOperationEmArea,
                           manualOperationCms := "ManualOperationControl_U1Em8".manualOperationCms,
                           Axis64Pos := "ManualOperationControl_U1Em8".axis,
                           AxisSoftCam := "ManualOperationControl_U1Em8".softCam,
                           twoWayAcutor := "ManualOperationControl_U1Em8".twoWayActuator,
                           Status := #StatusEm[8].Status,
                           errorID := #errorIDEm[8].errorID);
END_REGION

REGION Network 20 (SCL): Equipment Module 9 Cms Mapping
   REGION Input Mapping
       // TwoWayActuator
       "ManualOperationControl_U1Em9".twoWayActuator[1].monitoring := "Unit1.Em9.HmiInterface".cmVisionStageLiftUpDown.monitoring;
       "ManualOperationControl_U1Em9".twoWayActuator[2].monitoring := "Unit1.Em9.HmiInterface".cmVisionLightUpDown.monitoring;
   END_REGION


   REGION Output Mapping   
       // TwoWayActuator
       "Unit1.Em9.HmiInterface".cmVisionStageLiftUpDown.commands := "ManualOperationControl_U1Em9".twoWayActuator[1].commands;
       "Unit1.Em9.HmiInterface".cmVisionLightUpDown.commands := "ManualOperationControl_U1Em9".twoWayActuator[2].commands;
   END_REGION
END_REGION

REGION Network 21: Equipment Module 9
   RUNG wire#powerrail
      "CallManualOperationLines_EM"(disableUnit := #disableUnit1, manualOperationEm := "ManualOperationControl_U1Em9".manualOperationEm, manualOperationEmArea := "ManualOperationControl_U1Em9".manualOperationEmArea, manualOperationCms := "ManualOperationControl_U1Em9".manualOperationCms, Axis64Pos := "ManualOperationControl_U1Em9".axis, AxisSoftCam := "ManualOperationControl_U1Em9".softCam, twoWayAcutor := "ManualOperationControl_U1Em9".twoWayActuator, Status := #StatusEm[9].Status, errorID := #errorIDEm[9].errorID)
   END_RUNG
   // the same network as SCL:
   "CallManualOperationLines_EM"(disableUnit := #disableUnit1,
                           manualOperationEm := "ManualOperationControl_U1Em9".manualOperationEm,
                           manualOperationEmArea := "ManualOperationControl_U1Em9".manualOperationEmArea,
                           manualOperationCms := "ManualOperationControl_U1Em9".manualOperationCms,
                           Axis64Pos := "ManualOperationControl_U1Em9".axis,
                           AxisSoftCam := "ManualOperationControl_U1Em9".softCam,
                           twoWayAcutor := "ManualOperationControl_U1Em9".twoWayActuator,
                           Status := #StatusEm[9].Status,
                           errorID := #errorIDEm[9].errorID);
END_REGION

REGION Network 22 (SCL): Equipment Module 10 Cms Mapping
   REGION Input Mapping
       // TwoWayActuator
       "ManualOperationControl_U1Em10".twoWayActuator[1].monitoring := "Unit1.Em10.HmiInterface".cmLaserMarkCoverUpDown.monitoring;
       "ManualOperationControl_U1Em10".twoWayActuator[2].monitoring := "Unit1.Em10.HmiInterface".cmLaserMarkStageLiftUpDown.monitoring;
   END_REGION


   REGION Output Mapping 
       // TwoWayActuator
       "Unit1.Em10.HmiInterface".cmLaserMarkCoverUpDown.commands := "ManualOperationControl_U1Em10".twoWayActuator[1].commands;
       "Unit1.Em10.HmiInterface".cmLaserMarkStageLiftUpDown.commands := "ManualOperationControl_U1Em10".twoWayActuator[2].commands;
   END_REGION
END_REGION

REGION Network 23: Equipment Module 10
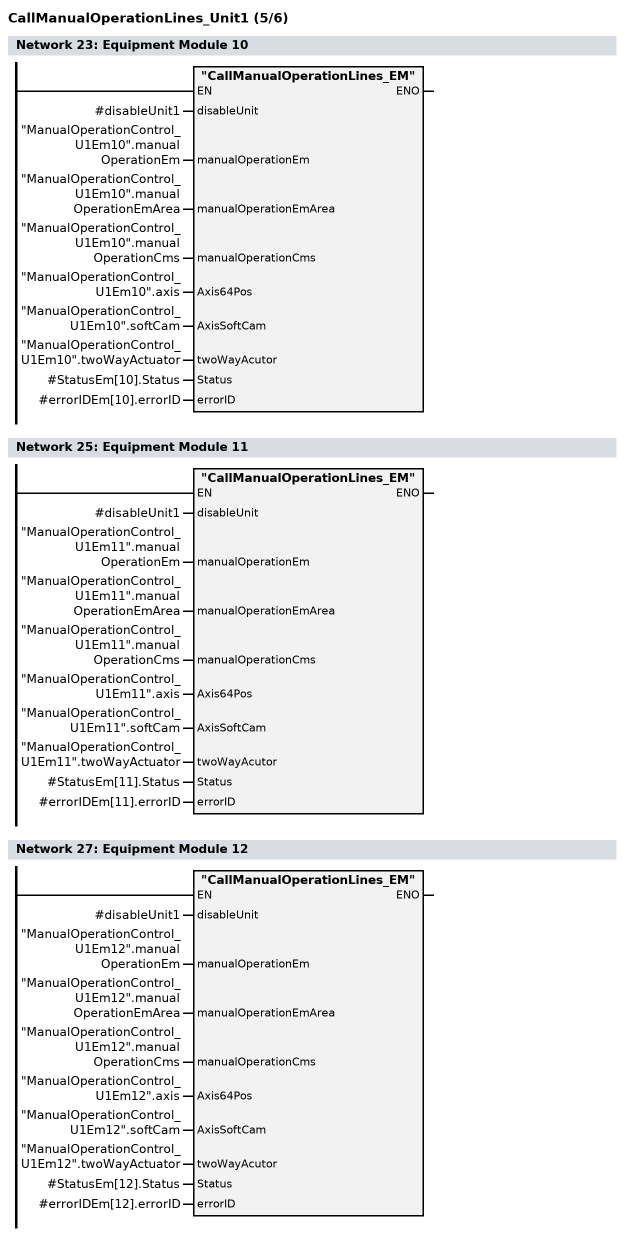
   RUNG wire#powerrail
      "CallManualOperationLines_EM"(disableUnit := #disableUnit1, manualOperationEm := "ManualOperationControl_U1Em10".manualOperationEm, manualOperationEmArea := "ManualOperationControl_U1Em10".manualOperationEmArea, manualOperationCms := "ManualOperationControl_U1Em10".manualOperationCms, Axis64Pos := "ManualOperationControl_U1Em10".axis, AxisSoftCam := "ManualOperationControl_U1Em10".softCam, twoWayAcutor := "ManualOperationControl_U1Em10".twoWayActuator, Status := #StatusEm[10].Status, errorID := #errorIDEm[10].errorID)
   END_RUNG
   // the same network as SCL:
   "CallManualOperationLines_EM"(disableUnit := #disableUnit1,
                           manualOperationEm := "ManualOperationControl_U1Em10".manualOperationEm,
                           manualOperationEmArea := "ManualOperationControl_U1Em10".manualOperationEmArea,
                           manualOperationCms := "ManualOperationControl_U1Em10".manualOperationCms,
                           Axis64Pos := "ManualOperationControl_U1Em10".axis,
                           AxisSoftCam := "ManualOperationControl_U1Em10".softCam,
                           twoWayAcutor := "ManualOperationControl_U1Em10".twoWayActuator,
                           Status := #StatusEm[10].Status,
                           errorID := #errorIDEm[10].errorID);
END_REGION

REGION Network 24 (SCL): Equipment Module 11 Cms Mapping
   REGION Input Mapping
       // TwoWayActuator
       "ManualOperationControl_U1Em11".twoWayActuator[1].monitoring := "Unit1.Em11.HmiInterface".cmWeightCheckStageLiftUpDown.monitoring;
   END_REGION


   REGION Output Mapping
       // TwoWayActuator
       "Unit1.Em11.HmiInterface".cmWeightCheckStageLiftUpDown.commands := "ManualOperationControl_U1Em11".twoWayActuator[1].commands;
   END_REGION
END_REGION

REGION Network 25: Equipment Module 11
   RUNG wire#powerrail
      "CallManualOperationLines_EM"(disableUnit := #disableUnit1, manualOperationEm := "ManualOperationControl_U1Em11".manualOperationEm, manualOperationEmArea := "ManualOperationControl_U1Em11".manualOperationEmArea, manualOperationCms := "ManualOperationControl_U1Em11".manualOperationCms, Axis64Pos := "ManualOperationControl_U1Em11".axis, AxisSoftCam := "ManualOperationControl_U1Em11".softCam, twoWayAcutor := "ManualOperationControl_U1Em11".twoWayActuator, Status := #StatusEm[11].Status, errorID := #errorIDEm[11].errorID)
   END_RUNG
   // the same network as SCL:
   "CallManualOperationLines_EM"(disableUnit := #disableUnit1,
                           manualOperationEm := "ManualOperationControl_U1Em11".manualOperationEm,
                           manualOperationEmArea := "ManualOperationControl_U1Em11".manualOperationEmArea,
                           manualOperationCms := "ManualOperationControl_U1Em11".manualOperationCms,
                           Axis64Pos := "ManualOperationControl_U1Em11".axis,
                           AxisSoftCam := "ManualOperationControl_U1Em11".softCam,
                           twoWayAcutor := "ManualOperationControl_U1Em11".twoWayActuator,
                           Status := #StatusEm[11].Status,
                           errorID := #errorIDEm[11].errorID);
END_REGION

REGION Network 26 (SCL): Equipment Module 12 Cms Mapping
   REGION Input Mapping
       // TwoWayActuator
       "ManualOperationControl_U1Em12".twoWayActuator[1].monitoring := "Unit1.Em12.HmiInterface".cmStackNgBoxClampMoverOpenClose.monitoring;
       "ManualOperationControl_U1Em12".twoWayActuator[2].monitoring := "Unit1.Em12.HmiInterface".cmStackNgBoxClampLeftOpenClose.monitoring;
       "ManualOperationControl_U1Em12".twoWayActuator[3].monitoring := "Unit1.Em12.HmiInterface".cmStackNgBoxClampRightOpenClose.monitoring;
       "ManualOperationControl_U1Em12".twoWayActuator[4].monitoring := "Unit1.Em12.HmiInterface".cmStackNgBoxLoadingUpDown.monitoring;
       "ManualOperationControl_U1Em12".twoWayActuator[5].monitoring := "Unit1.Em12.HmiInterface".cmStackNgBoxUnitMoverBwdFwd.monitoring;
       "ManualOperationControl_U1Em12".twoWayActuator[6].monitoring := "Unit1.Em12.HmiInterface".cmStackNgBoxLiftDownUp.monitoring;
       "ManualOperationControl_U1Em12".twoWayActuator[7].monitoring := "Unit1.Em12.HmiInterface".cmStackNgBoxLockDownUp.monitoring;
   END_REGION


   REGION Output Mapping
       // TwoWayActuator
       "Unit1.Em12.HmiInterface".cmStackNgBoxClampMoverOpenClose.commands := "ManualOperationControl_U1Em12".twoWayActuator[1].commands;
       "Unit1.Em12.HmiInterface".cmStackNgBoxClampLeftOpenClose.commands := "ManualOperationControl_U1Em12".twoWayActuator[2].commands;
       "Unit1.Em12.HmiInterface".cmStackNgBoxClampRightOpenClose.commands := "ManualOperationControl_U1Em12".twoWayActuator[3].commands;
       "Unit1.Em12.HmiInterface".cmStackNgBoxLoadingUpDown.commands := "ManualOperationControl_U1Em12".twoWayActuator[4].commands;
       "Unit1.Em12.HmiInterface".cmStackNgBoxUnitMoverBwdFwd.commands := "ManualOperationControl_U1Em12".twoWayActuator[5].commands;
       "Unit1.Em12.HmiInterface".cmStackNgBoxLiftDownUp.commands := "ManualOperationControl_U1Em12".twoWayActuator[6].commands;
       "Unit1.Em12.HmiInterface".cmStackNgBoxLockDownUp.commands := "ManualOperationControl_U1Em12".twoWayActuator[7].commands;
   END_REGION
END_REGION

REGION Network 27: Equipment Module 12
   RUNG wire#powerrail
      "CallManualOperationLines_EM"(disableUnit := #disableUnit1, manualOperationEm := "ManualOperationControl_U1Em12".manualOperationEm, manualOperationEmArea := "ManualOperationControl_U1Em12".manualOperationEmArea, manualOperationCms := "ManualOperationControl_U1Em12".manualOperationCms, Axis64Pos := "ManualOperationControl_U1Em12".axis, AxisSoftCam := "ManualOperationControl_U1Em12".softCam, twoWayAcutor := "ManualOperationControl_U1Em12".twoWayActuator, Status := #StatusEm[12].Status, errorID := #errorIDEm[12].errorID)
   END_RUNG
   // the same network as SCL:
   "CallManualOperationLines_EM"(disableUnit := #disableUnit1,
                           manualOperationEm := "ManualOperationControl_U1Em12".manualOperationEm,
                           manualOperationEmArea := "ManualOperationControl_U1Em12".manualOperationEmArea,
                           manualOperationCms := "ManualOperationControl_U1Em12".manualOperationCms,
                           Axis64Pos := "ManualOperationControl_U1Em12".axis,
                           AxisSoftCam := "ManualOperationControl_U1Em12".softCam,
                           twoWayAcutor := "ManualOperationControl_U1Em12".twoWayActuator,
                           Status := #StatusEm[12].Status,
                           errorID := #errorIDEm[12].errorID);
END_REGION

REGION Network 28 (SCL): Equipment Module 13 Cms Mapping
   REGION Input Mapping
        // Axis
       "ManualOperationControl_U1Em13".axis[1].monitoring := "Unit1.Em13.HmiInterface".cmJRUnloadingPnPAxisX.monitoring;
       "ManualOperationControl_U1Em13".axis[2].monitoring := "Unit1.Em13.HmiInterface".cmJRUnloadingPnPAxisZ.monitoring;
       "ManualOperationControl_U1Em13".axis[3].monitoring := "Unit1.Em13.HmiInterface".cmJRUnloadingPnPAxisC.monitoring;

       // SoftCam
       "ManualOperationControl_U1Em13".softCam[1] := "Unit1.Em13.HmiInterface".cm.softcam.jrUnIoadingPnPAxisX;
       "ManualOperationControl_U1Em13".softCam[2] := "Unit1.Em13.HmiInterface".cm.softcam.jrUnIoadingPnPAxisZ;
       "ManualOperationControl_U1Em13".softCam[3] := "Unit1.Em13.HmiInterface".cm.softcam.jrUnIoadingPnPAxisC;

       // TwoWayActuator
       "ManualOperationControl_U1Em13".twoWayActuator[1].monitoring := "Unit1.Em13.HmiInterface".cmJRUnloadingPnPClampOpenClose.monitoring;
   END_REGION


   REGION Output Mapping
       // Axis
       "Unit1.Em13.HmiInterface".cmJRUnloadingPnPAxisX.commands.jogForward := "ManualOperationControl_U1Em13".axis[1].commands.jogForward;
       "Unit1.Em13.HmiInterface".cmJRUnloadingPnPAxisX.commands.jogBackward := "ManualOperationControl_U1Em13".axis[1].commands.jogBackward;
       "Unit1.Em13.HmiInterface".cmJRUnloadingPnPAxisZ.commands.jogForward := "ManualOperationControl_U1Em13".axis[2].commands.jogForward;
       "Unit1.Em13.HmiInterface".cmJRUnloadingPnPAxisZ.commands.jogBackward := "ManualOperationControl_U1Em13".axis[2].commands.jogBackward;
       "Unit1.Em13.HmiInterface".cmJRUnloadingPnPAxisC.commands.jogForward := "ManualOperationControl_U1Em13".axis[3].commands.jogForward;
       "Unit1.Em13.HmiInterface".cmJRUnloadingPnPAxisC.commands.jogBackward := "ManualOperationControl_U1Em13".axis[3].commands.jogBackward;

       // TwoWayActuator
       "Unit1.Em13.HmiInterface".cmJRUnloadingPnPClampOpenClose.commands := "ManualOperationControl_U1Em13".twoWayActuator[1].commands;
   END_REGION
END_REGION

REGION Network 29: Equipment Module 13
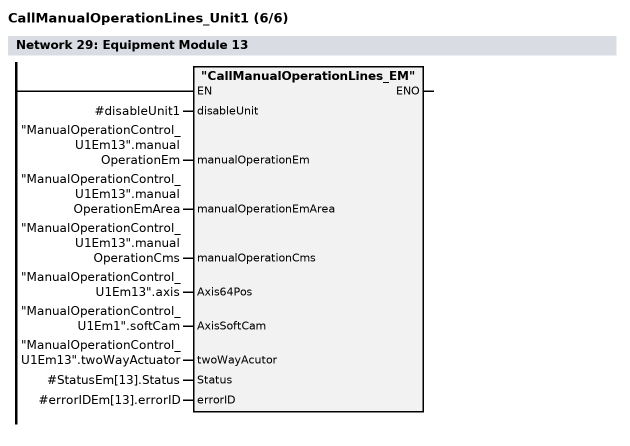
   RUNG wire#powerrail
      "CallManualOperationLines_EM"(disableUnit := #disableUnit1, manualOperationEm := "ManualOperationControl_U1Em13".manualOperationEm, manualOperationEmArea := "ManualOperationControl_U1Em13".manualOperationEmArea, manualOperationCms := "ManualOperationControl_U1Em13".manualOperationCms, Axis64Pos := "ManualOperationControl_U1Em13".axis, AxisSoftCam := "ManualOperationControl_U1Em1".softCam, twoWayAcutor := "ManualOperationControl_U1Em13".twoWayActuator, Status := #StatusEm[13].Status, errorID := #errorIDEm[13].errorID)
   END_RUNG
   // the same network as SCL:
   "CallManualOperationLines_EM"(disableUnit := #disableUnit1,
                           manualOperationEm := "ManualOperationControl_U1Em13".manualOperationEm,
                           manualOperationEmArea := "ManualOperationControl_U1Em13".manualOperationEmArea,
                           manualOperationCms := "ManualOperationControl_U1Em13".manualOperationCms,
                           Axis64Pos := "ManualOperationControl_U1Em13".axis,
                           AxisSoftCam := "ManualOperationControl_U1Em1".softCam,
                           twoWayAcutor := "ManualOperationControl_U1Em13".twoWayActuator,
                           Status := #StatusEm[13].Status,
                           errorID := #errorIDEm[13].errorID);
END_REGION
END_FUNCTION

FUNCTION "CallManualOperationLines_EM" : Void   // FC82, LAD
// stored: SetENOAutomatically false
   VAR_INPUT
      disableUnit : Bool;
   END_VAR
   VAR_IN_OUT
      manualOperationEm : "LAF_typeManEm";
      manualOperationEmArea : Array[*] of "LAF_typeManOperationArea";
      manualOperationCms : Array[*] of "LAF_typeManOperation";
      Axis64Pos : Array[*] of "LBC_typeAxis64PosInterface";
      AxisSoftCam : Array[*] of "LER_typeSoftCamRelation";
      twoWayAcutor : Array[*] of "LBC_typeTwoWayActuatorInterface";
      Status : Array[*] of Word;
      errorID : Array[*] of Word;
   END_VAR
   VAR_TEMP
      tempLowerBoundAxis : Int;
      tempUpperBoundAxis : Int;
      tempLowerBoundTwoWayAct : Int;
      tempUpperBoundTwoWayAct : Int;
      tempEnd : Bool;
   END_VAR
BEGIN

REGION Network 1: Detect lower and upper bound of the array for further processing
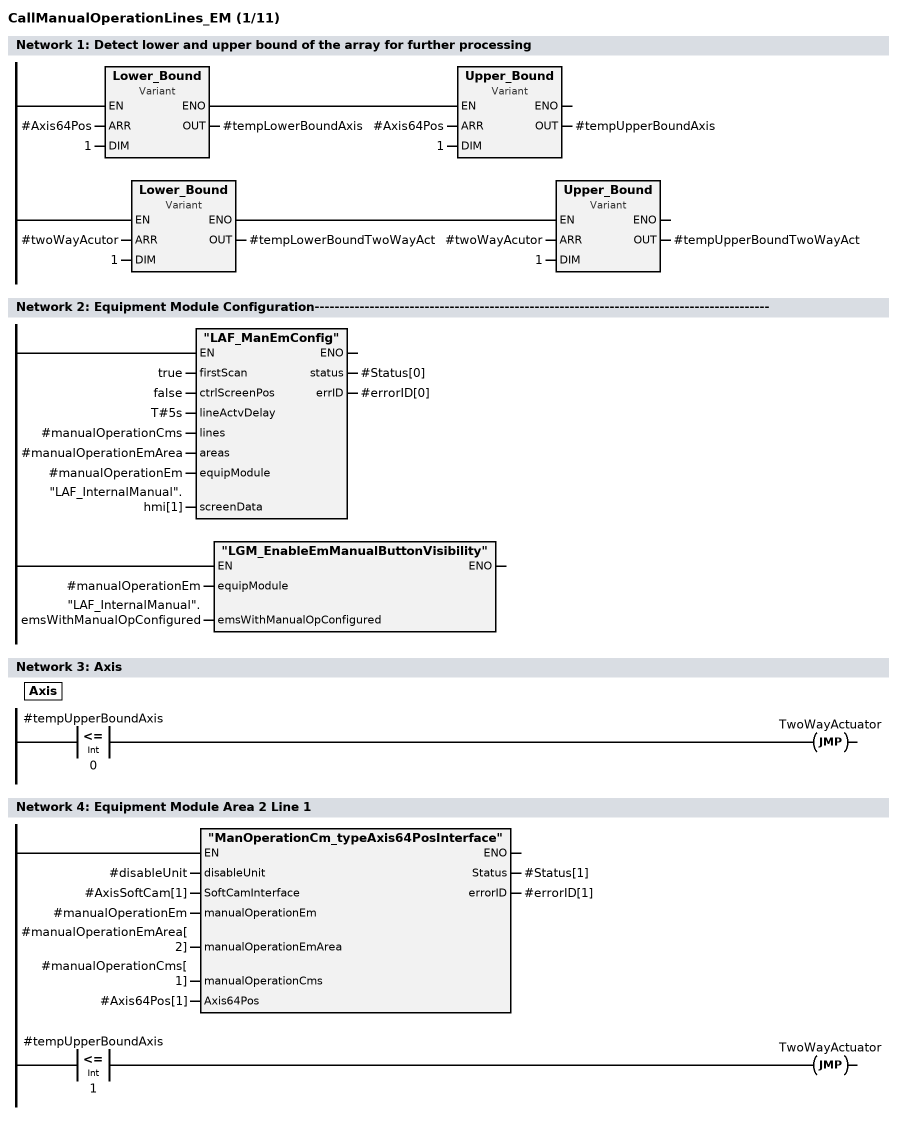
   // no SCL statement known for Lower_Bound, Upper_Bound: written as a call
   // ENO of a box is taken as its EN; it also drops when the box reports an error
   Lower_Bound(arr := #Axis64Pos, dim := 1, out => #tempLowerBoundAxis);
   Upper_Bound(arr := #Axis64Pos, dim := 1, out => #tempUpperBoundAxis);
   Lower_Bound(arr := #twoWayAcutor, dim := 1, out => #tempLowerBoundTwoWayAct);
   Upper_Bound(arr := #twoWayAcutor, dim := 1, out => #tempUpperBoundTwoWayAct);
END_REGION

REGION Network 2: Equipment Module Configuration-------------------------------------------------------------------------------------------
   RUNG wire#powerrail
      "LAF_ManEmConfig"(firstScan := true, ctrlScreenPos := false, lineActvDelay := T#5s, lines := #manualOperationCms, areas := #manualOperationEmArea, equipModule := #manualOperationEm, screenData := "LAF_InternalManual".hmi[1], status => #Status[0], errID => #errorID[0])
   END_RUNG
   RUNG wire#powerrail
      "LGM_EnableEmManualButtonVisibility"(equipModule := #manualOperationEm, emsWithManualOpConfigured := "LAF_InternalManual".emsWithManualOpConfigured)
   END_RUNG
   // the same network as SCL:
   "LAF_ManEmConfig"(firstScan := true,
                     ctrlScreenPos := false,
                     lineActvDelay := T#5s,
                     lines := #manualOperationCms,
                     areas := #manualOperationEmArea,
                     equipModule := #manualOperationEm,
                     screenData := "LAF_InternalManual".hmi[1],
                     status => #Status[0],
                     errID => #errorID[0]);
   "LGM_EnableEmManualButtonVisibility"(equipModule := #manualOperationEm,
                           emsWithManualOpConfigured := "LAF_InternalManual".emsWithManualOpConfigured);
END_REGION

REGION Network 3: Axis
   Label( Axis )
   RUNG wire#powerrail
      { S7_Templates := "SrcType := Int" } LE_Contact(in1 := #tempUpperBoundAxis, in2 := 0)
      JumpCoil( TwoWayActuator )
   END_RUNG
   // the same network as SCL:
   Axis:
   IF #tempUpperBoundAxis <= 0 THEN GOTO TwoWayActuator; END_IF;
END_REGION

REGION Network 4: Equipment Module Area 2 Line 1
   RUNG wire#powerrail
      "ManOperationCm_typeAxis64PosInterface"(disableUnit := #disableUnit, SoftCamInterface := #AxisSoftCam[1], manualOperationEm := #manualOperationEm, manualOperationEmArea := #manualOperationEmArea[2], manualOperationCms := #manualOperationCms[1], Axis64Pos := #Axis64Pos[1], Status => #Status[1], errorID => #errorID[1])
   END_RUNG
   RUNG wire#powerrail
      { S7_Templates := "SrcType := Int" } LE_Contact(in1 := #tempUpperBoundAxis, in2 := 1)
      JumpCoil( TwoWayActuator )
   END_RUNG
   // the same network as SCL:
   "ManOperationCm_typeAxis64PosInterface"(disableUnit := #disableUnit,
                           SoftCamInterface := #AxisSoftCam[1],
                           manualOperationEm := #manualOperationEm,
                           manualOperationEmArea := #manualOperationEmArea[2],
                           manualOperationCms := #manualOperationCms[1],
                           Axis64Pos := #Axis64Pos[1],
                           Status => #Status[1],
                           errorID => #errorID[1]);
   IF #tempUpperBoundAxis <= 1 THEN GOTO TwoWayActuator; END_IF;
END_REGION

REGION Network 5: Equipment Module Area 2 Line 2
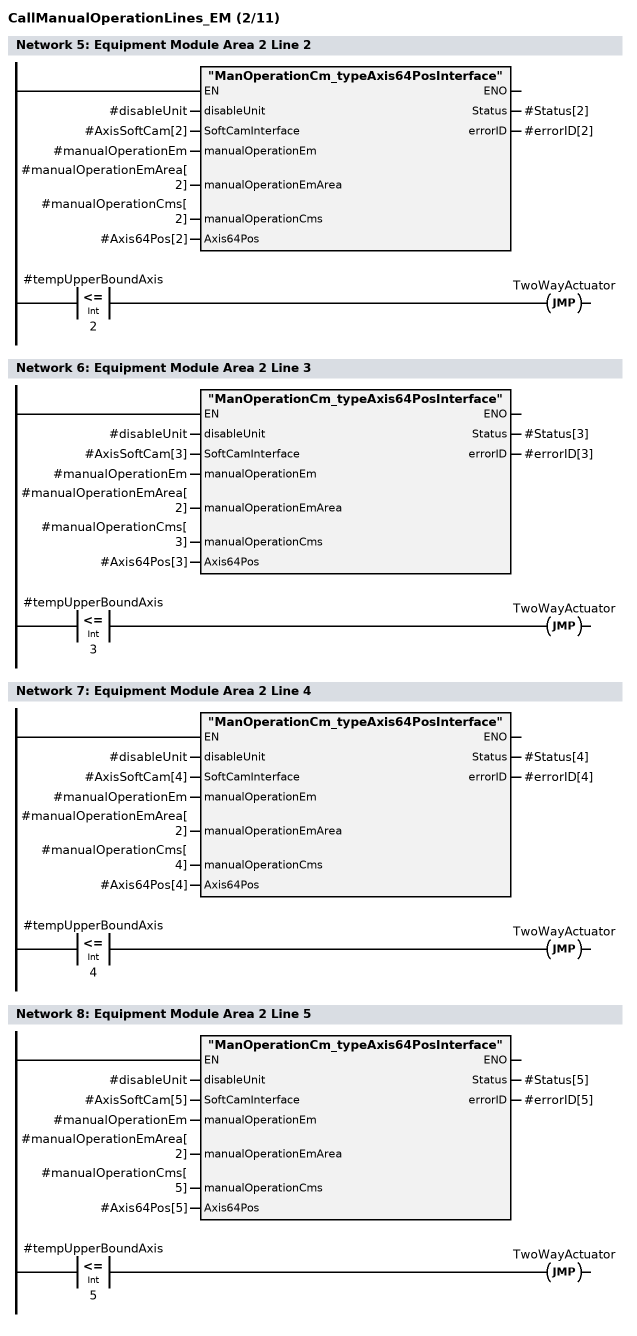
   RUNG wire#powerrail
      "ManOperationCm_typeAxis64PosInterface"(disableUnit := #disableUnit, SoftCamInterface := #AxisSoftCam[2], manualOperationEm := #manualOperationEm, manualOperationEmArea := #manualOperationEmArea[2], manualOperationCms := #manualOperationCms[2], Axis64Pos := #Axis64Pos[2], Status => #Status[2], errorID => #errorID[2])
   END_RUNG
   RUNG wire#powerrail
      { S7_Templates := "SrcType := Int" } LE_Contact(in1 := #tempUpperBoundAxis, in2 := 2)
      JumpCoil( TwoWayActuator )
   END_RUNG
   // the same network as SCL:
   "ManOperationCm_typeAxis64PosInterface"(disableUnit := #disableUnit,
                           SoftCamInterface := #AxisSoftCam[2],
                           manualOperationEm := #manualOperationEm,
                           manualOperationEmArea := #manualOperationEmArea[2],
                           manualOperationCms := #manualOperationCms[2],
                           Axis64Pos := #Axis64Pos[2],
                           Status => #Status[2],
                           errorID => #errorID[2]);
   IF #tempUpperBoundAxis <= 2 THEN GOTO TwoWayActuator; END_IF;
END_REGION

REGION Network 6: Equipment Module Area 2 Line 3
   RUNG wire#powerrail
      "ManOperationCm_typeAxis64PosInterface"(disableUnit := #disableUnit, SoftCamInterface := #AxisSoftCam[3], manualOperationEm := #manualOperationEm, manualOperationEmArea := #manualOperationEmArea[2], manualOperationCms := #manualOperationCms[3], Axis64Pos := #Axis64Pos[3], Status => #Status[3], errorID => #errorID[3])
   END_RUNG
   RUNG wire#powerrail
      { S7_Templates := "SrcType := Int" } LE_Contact(in1 := #tempUpperBoundAxis, in2 := 3)
      JumpCoil( TwoWayActuator )
   END_RUNG
   // the same network as SCL:
   "ManOperationCm_typeAxis64PosInterface"(disableUnit := #disableUnit,
                           SoftCamInterface := #AxisSoftCam[3],
                           manualOperationEm := #manualOperationEm,
                           manualOperationEmArea := #manualOperationEmArea[2],
                           manualOperationCms := #manualOperationCms[3],
                           Axis64Pos := #Axis64Pos[3],
                           Status => #Status[3],
                           errorID => #errorID[3]);
   IF #tempUpperBoundAxis <= 3 THEN GOTO TwoWayActuator; END_IF;
END_REGION

REGION Network 7: Equipment Module Area 2 Line 4
   RUNG wire#powerrail
      "ManOperationCm_typeAxis64PosInterface"(disableUnit := #disableUnit, SoftCamInterface := #AxisSoftCam[4], manualOperationEm := #manualOperationEm, manualOperationEmArea := #manualOperationEmArea[2], manualOperationCms := #manualOperationCms[4], Axis64Pos := #Axis64Pos[4], Status => #Status[4], errorID => #errorID[4])
   END_RUNG
   RUNG wire#powerrail
      { S7_Templates := "SrcType := Int" } LE_Contact(in1 := #tempUpperBoundAxis, in2 := 4)
      JumpCoil( TwoWayActuator )
   END_RUNG
   // the same network as SCL:
   "ManOperationCm_typeAxis64PosInterface"(disableUnit := #disableUnit,
                           SoftCamInterface := #AxisSoftCam[4],
                           manualOperationEm := #manualOperationEm,
                           manualOperationEmArea := #manualOperationEmArea[2],
                           manualOperationCms := #manualOperationCms[4],
                           Axis64Pos := #Axis64Pos[4],
                           Status => #Status[4],
                           errorID => #errorID[4]);
   IF #tempUpperBoundAxis <= 4 THEN GOTO TwoWayActuator; END_IF;
END_REGION

REGION Network 8: Equipment Module Area 2 Line 5
   RUNG wire#powerrail
      "ManOperationCm_typeAxis64PosInterface"(disableUnit := #disableUnit, SoftCamInterface := #AxisSoftCam[5], manualOperationEm := #manualOperationEm, manualOperationEmArea := #manualOperationEmArea[2], manualOperationCms := #manualOperationCms[5], Axis64Pos := #Axis64Pos[5], Status => #Status[5], errorID => #errorID[5])
   END_RUNG
   RUNG wire#powerrail
      { S7_Templates := "SrcType := Int" } LE_Contact(in1 := #tempUpperBoundAxis, in2 := 5)
      JumpCoil( TwoWayActuator )
   END_RUNG
   // the same network as SCL:
   "ManOperationCm_typeAxis64PosInterface"(disableUnit := #disableUnit,
                           SoftCamInterface := #AxisSoftCam[5],
                           manualOperationEm := #manualOperationEm,
                           manualOperationEmArea := #manualOperationEmArea[2],
                           manualOperationCms := #manualOperationCms[5],
                           Axis64Pos := #Axis64Pos[5],
                           Status => #Status[5],
                           errorID => #errorID[5]);
   IF #tempUpperBoundAxis <= 5 THEN GOTO TwoWayActuator; END_IF;
END_REGION

REGION Network 9: Equipment Module Area 2 Line 6
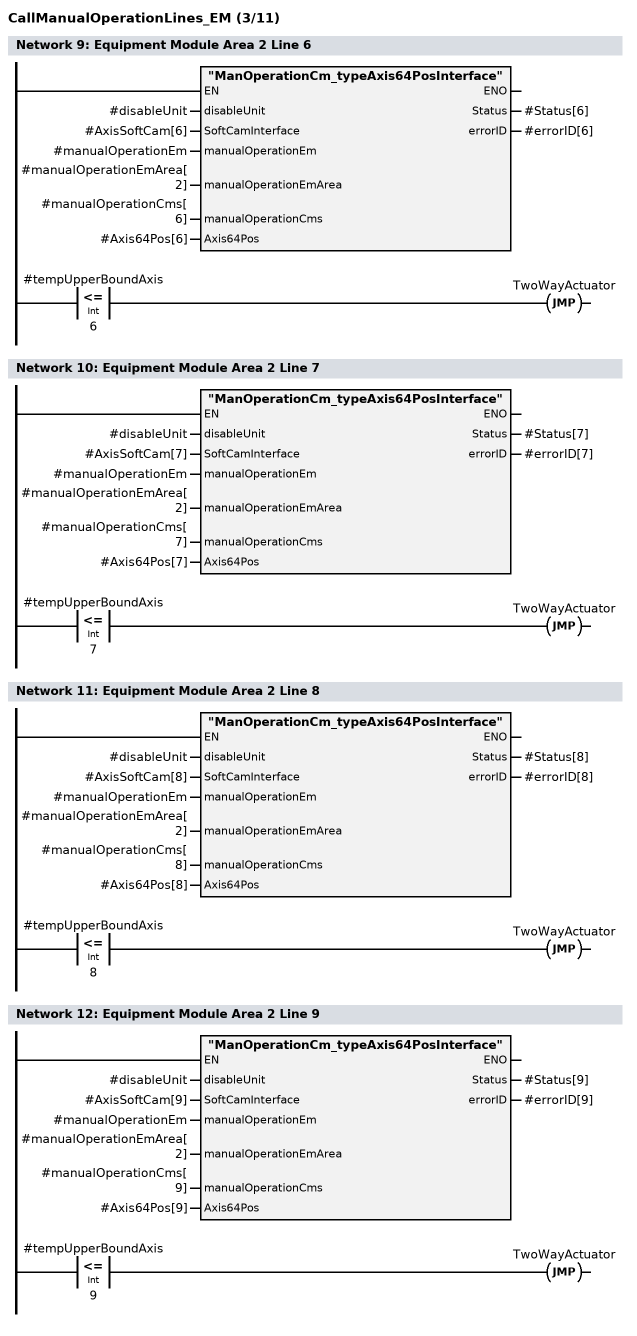
   RUNG wire#powerrail
      "ManOperationCm_typeAxis64PosInterface"(disableUnit := #disableUnit, SoftCamInterface := #AxisSoftCam[6], manualOperationEm := #manualOperationEm, manualOperationEmArea := #manualOperationEmArea[2], manualOperationCms := #manualOperationCms[6], Axis64Pos := #Axis64Pos[6], Status => #Status[6], errorID => #errorID[6])
   END_RUNG
   RUNG wire#powerrail
      { S7_Templates := "SrcType := Int" } LE_Contact(in1 := #tempUpperBoundAxis, in2 := 6)
      JumpCoil( TwoWayActuator )
   END_RUNG
   // the same network as SCL:
   "ManOperationCm_typeAxis64PosInterface"(disableUnit := #disableUnit,
                           SoftCamInterface := #AxisSoftCam[6],
                           manualOperationEm := #manualOperationEm,
                           manualOperationEmArea := #manualOperationEmArea[2],
                           manualOperationCms := #manualOperationCms[6],
                           Axis64Pos := #Axis64Pos[6],
                           Status => #Status[6],
                           errorID => #errorID[6]);
   IF #tempUpperBoundAxis <= 6 THEN GOTO TwoWayActuator; END_IF;
END_REGION

REGION Network 10: Equipment Module Area 2 Line 7
   RUNG wire#powerrail
      "ManOperationCm_typeAxis64PosInterface"(disableUnit := #disableUnit, SoftCamInterface := #AxisSoftCam[7], manualOperationEm := #manualOperationEm, manualOperationEmArea := #manualOperationEmArea[2], manualOperationCms := #manualOperationCms[7], Axis64Pos := #Axis64Pos[7], Status => #Status[7], errorID => #errorID[7])
   END_RUNG
   RUNG wire#powerrail
      { S7_Templates := "SrcType := Int" } LE_Contact(in1 := #tempUpperBoundAxis, in2 := 7)
      JumpCoil( TwoWayActuator )
   END_RUNG
   // the same network as SCL:
   "ManOperationCm_typeAxis64PosInterface"(disableUnit := #disableUnit,
                           SoftCamInterface := #AxisSoftCam[7],
                           manualOperationEm := #manualOperationEm,
                           manualOperationEmArea := #manualOperationEmArea[2],
                           manualOperationCms := #manualOperationCms[7],
                           Axis64Pos := #Axis64Pos[7],
                           Status => #Status[7],
                           errorID => #errorID[7]);
   IF #tempUpperBoundAxis <= 7 THEN GOTO TwoWayActuator; END_IF;
END_REGION

REGION Network 11: Equipment Module Area 2 Line 8
   RUNG wire#powerrail
      "ManOperationCm_typeAxis64PosInterface"(disableUnit := #disableUnit, SoftCamInterface := #AxisSoftCam[8], manualOperationEm := #manualOperationEm, manualOperationEmArea := #manualOperationEmArea[2], manualOperationCms := #manualOperationCms[8], Axis64Pos := #Axis64Pos[8], Status => #Status[8], errorID => #errorID[8])
   END_RUNG
   RUNG wire#powerrail
      { S7_Templates := "SrcType := Int" } LE_Contact(in1 := #tempUpperBoundAxis, in2 := 8)
      JumpCoil( TwoWayActuator )
   END_RUNG
   // the same network as SCL:
   "ManOperationCm_typeAxis64PosInterface"(disableUnit := #disableUnit,
                           SoftCamInterface := #AxisSoftCam[8],
                           manualOperationEm := #manualOperationEm,
                           manualOperationEmArea := #manualOperationEmArea[2],
                           manualOperationCms := #manualOperationCms[8],
                           Axis64Pos := #Axis64Pos[8],
                           Status => #Status[8],
                           errorID => #errorID[8]);
   IF #tempUpperBoundAxis <= 8 THEN GOTO TwoWayActuator; END_IF;
END_REGION

REGION Network 12: Equipment Module Area 2 Line 9
   RUNG wire#powerrail
      "ManOperationCm_typeAxis64PosInterface"(disableUnit := #disableUnit, SoftCamInterface := #AxisSoftCam[9], manualOperationEm := #manualOperationEm, manualOperationEmArea := #manualOperationEmArea[2], manualOperationCms := #manualOperationCms[9], Axis64Pos := #Axis64Pos[9], Status => #Status[9], errorID => #errorID[9])
   END_RUNG
   RUNG wire#powerrail
      { S7_Templates := "SrcType := Int" } LE_Contact(in1 := #tempUpperBoundAxis, in2 := 9)
      JumpCoil( TwoWayActuator )
   END_RUNG
   // the same network as SCL:
   "ManOperationCm_typeAxis64PosInterface"(disableUnit := #disableUnit,
                           SoftCamInterface := #AxisSoftCam[9],
                           manualOperationEm := #manualOperationEm,
                           manualOperationEmArea := #manualOperationEmArea[2],
                           manualOperationCms := #manualOperationCms[9],
                           Axis64Pos := #Axis64Pos[9],
                           Status => #Status[9],
                           errorID => #errorID[9]);
   IF #tempUpperBoundAxis <= 9 THEN GOTO TwoWayActuator; END_IF;
END_REGION

REGION Network 13: Equipment Module Area 2 Line 10
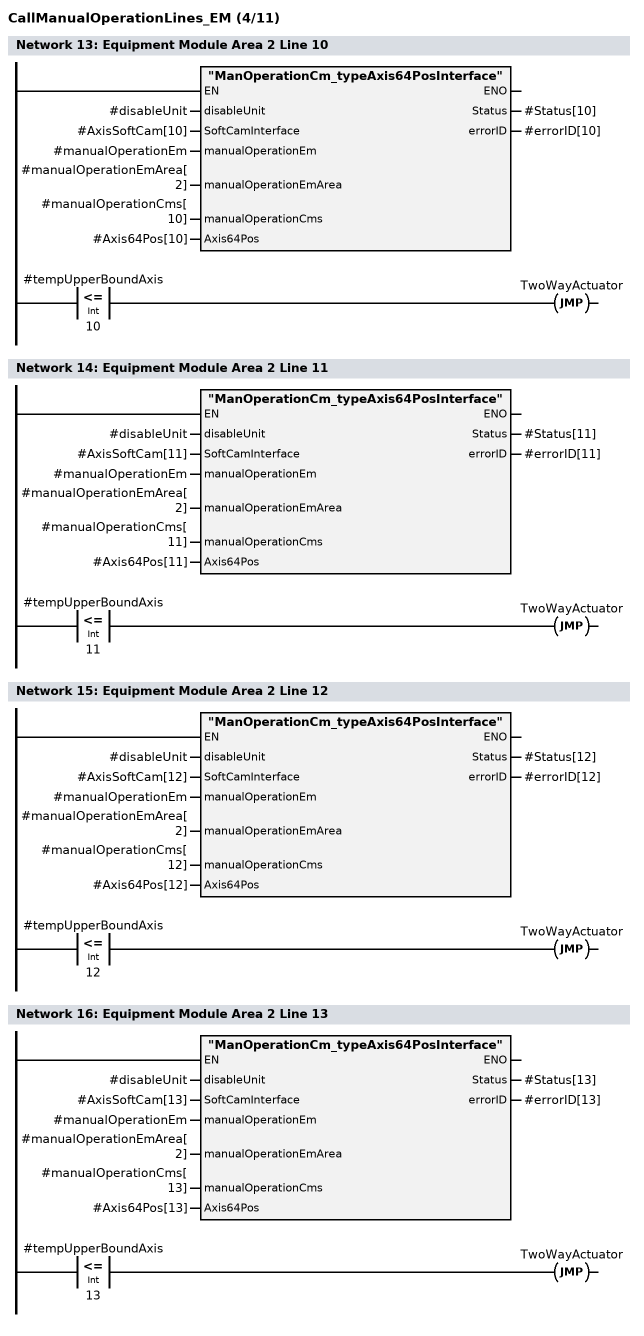
   RUNG wire#powerrail
      "ManOperationCm_typeAxis64PosInterface"(disableUnit := #disableUnit, SoftCamInterface := #AxisSoftCam[10], manualOperationEm := #manualOperationEm, manualOperationEmArea := #manualOperationEmArea[2], manualOperationCms := #manualOperationCms[10], Axis64Pos := #Axis64Pos[10], Status => #Status[10], errorID => #errorID[10])
   END_RUNG
   RUNG wire#powerrail
      { S7_Templates := "SrcType := Int" } LE_Contact(in1 := #tempUpperBoundAxis, in2 := 10)
      JumpCoil( TwoWayActuator )
   END_RUNG
   // the same network as SCL:
   "ManOperationCm_typeAxis64PosInterface"(disableUnit := #disableUnit,
                           SoftCamInterface := #AxisSoftCam[10],
                           manualOperationEm := #manualOperationEm,
                           manualOperationEmArea := #manualOperationEmArea[2],
                           manualOperationCms := #manualOperationCms[10],
                           Axis64Pos := #Axis64Pos[10],
                           Status => #Status[10],
                           errorID => #errorID[10]);
   IF #tempUpperBoundAxis <= 10 THEN GOTO TwoWayActuator; END_IF;
END_REGION

REGION Network 14: Equipment Module Area 2 Line 11
   RUNG wire#powerrail
      "ManOperationCm_typeAxis64PosInterface"(disableUnit := #disableUnit, SoftCamInterface := #AxisSoftCam[11], manualOperationEm := #manualOperationEm, manualOperationEmArea := #manualOperationEmArea[2], manualOperationCms := #manualOperationCms[11], Axis64Pos := #Axis64Pos[11], Status => #Status[11], errorID => #errorID[11])
   END_RUNG
   RUNG wire#powerrail
      { S7_Templates := "SrcType := Int" } LE_Contact(in1 := #tempUpperBoundAxis, in2 := 11)
      JumpCoil( TwoWayActuator )
   END_RUNG
   // the same network as SCL:
   "ManOperationCm_typeAxis64PosInterface"(disableUnit := #disableUnit,
                           SoftCamInterface := #AxisSoftCam[11],
                           manualOperationEm := #manualOperationEm,
                           manualOperationEmArea := #manualOperationEmArea[2],
                           manualOperationCms := #manualOperationCms[11],
                           Axis64Pos := #Axis64Pos[11],
                           Status => #Status[11],
                           errorID => #errorID[11]);
   IF #tempUpperBoundAxis <= 11 THEN GOTO TwoWayActuator; END_IF;
END_REGION

REGION Network 15: Equipment Module Area 2 Line 12
   RUNG wire#powerrail
      "ManOperationCm_typeAxis64PosInterface"(disableUnit := #disableUnit, SoftCamInterface := #AxisSoftCam[12], manualOperationEm := #manualOperationEm, manualOperationEmArea := #manualOperationEmArea[2], manualOperationCms := #manualOperationCms[12], Axis64Pos := #Axis64Pos[12], Status => #Status[12], errorID => #errorID[12])
   END_RUNG
   RUNG wire#powerrail
      { S7_Templates := "SrcType := Int" } LE_Contact(in1 := #tempUpperBoundAxis, in2 := 12)
      JumpCoil( TwoWayActuator )
   END_RUNG
   // the same network as SCL:
   "ManOperationCm_typeAxis64PosInterface"(disableUnit := #disableUnit,
                           SoftCamInterface := #AxisSoftCam[12],
                           manualOperationEm := #manualOperationEm,
                           manualOperationEmArea := #manualOperationEmArea[2],
                           manualOperationCms := #manualOperationCms[12],
                           Axis64Pos := #Axis64Pos[12],
                           Status => #Status[12],
                           errorID => #errorID[12]);
   IF #tempUpperBoundAxis <= 12 THEN GOTO TwoWayActuator; END_IF;
END_REGION

REGION Network 16: Equipment Module Area 2 Line 13
   RUNG wire#powerrail
      "ManOperationCm_typeAxis64PosInterface"(disableUnit := #disableUnit, SoftCamInterface := #AxisSoftCam[13], manualOperationEm := #manualOperationEm, manualOperationEmArea := #manualOperationEmArea[2], manualOperationCms := #manualOperationCms[13], Axis64Pos := #Axis64Pos[13], Status => #Status[13], errorID => #errorID[13])
   END_RUNG
   RUNG wire#powerrail
      { S7_Templates := "SrcType := Int" } LE_Contact(in1 := #tempUpperBoundAxis, in2 := 13)
      JumpCoil( TwoWayActuator )
   END_RUNG
   // the same network as SCL:
   "ManOperationCm_typeAxis64PosInterface"(disableUnit := #disableUnit,
                           SoftCamInterface := #AxisSoftCam[13],
                           manualOperationEm := #manualOperationEm,
                           manualOperationEmArea := #manualOperationEmArea[2],
                           manualOperationCms := #manualOperationCms[13],
                           Axis64Pos := #Axis64Pos[13],
                           Status => #Status[13],
                           errorID => #errorID[13]);
   IF #tempUpperBoundAxis <= 13 THEN GOTO TwoWayActuator; END_IF;
END_REGION

REGION Network 17: Equipment Module Area 2 Line 14
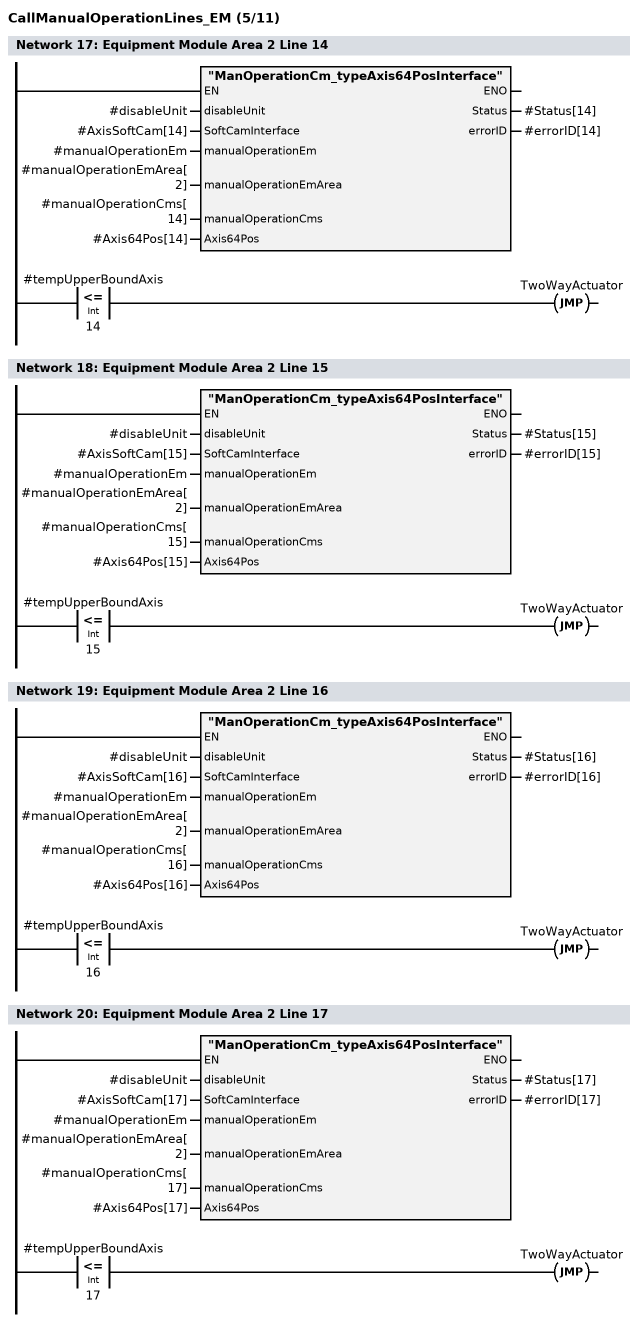
   RUNG wire#powerrail
      "ManOperationCm_typeAxis64PosInterface"(disableUnit := #disableUnit, SoftCamInterface := #AxisSoftCam[14], manualOperationEm := #manualOperationEm, manualOperationEmArea := #manualOperationEmArea[2], manualOperationCms := #manualOperationCms[14], Axis64Pos := #Axis64Pos[14], Status => #Status[14], errorID => #errorID[14])
   END_RUNG
   RUNG wire#powerrail
      { S7_Templates := "SrcType := Int" } LE_Contact(in1 := #tempUpperBoundAxis, in2 := 14)
      JumpCoil( TwoWayActuator )
   END_RUNG
   // the same network as SCL:
   "ManOperationCm_typeAxis64PosInterface"(disableUnit := #disableUnit,
                           SoftCamInterface := #AxisSoftCam[14],
                           manualOperationEm := #manualOperationEm,
                           manualOperationEmArea := #manualOperationEmArea[2],
                           manualOperationCms := #manualOperationCms[14],
                           Axis64Pos := #Axis64Pos[14],
                           Status => #Status[14],
                           errorID => #errorID[14]);
   IF #tempUpperBoundAxis <= 14 THEN GOTO TwoWayActuator; END_IF;
END_REGION

REGION Network 18: Equipment Module Area 2 Line 15
   RUNG wire#powerrail
      "ManOperationCm_typeAxis64PosInterface"(disableUnit := #disableUnit, SoftCamInterface := #AxisSoftCam[15], manualOperationEm := #manualOperationEm, manualOperationEmArea := #manualOperationEmArea[2], manualOperationCms := #manualOperationCms[15], Axis64Pos := #Axis64Pos[15], Status => #Status[15], errorID => #errorID[15])
   END_RUNG
   RUNG wire#powerrail
      { S7_Templates := "SrcType := Int" } LE_Contact(in1 := #tempUpperBoundAxis, in2 := 15)
      JumpCoil( TwoWayActuator )
   END_RUNG
   // the same network as SCL:
   "ManOperationCm_typeAxis64PosInterface"(disableUnit := #disableUnit,
                           SoftCamInterface := #AxisSoftCam[15],
                           manualOperationEm := #manualOperationEm,
                           manualOperationEmArea := #manualOperationEmArea[2],
                           manualOperationCms := #manualOperationCms[15],
                           Axis64Pos := #Axis64Pos[15],
                           Status => #Status[15],
                           errorID => #errorID[15]);
   IF #tempUpperBoundAxis <= 15 THEN GOTO TwoWayActuator; END_IF;
END_REGION

REGION Network 19: Equipment Module Area 2 Line 16
   RUNG wire#powerrail
      "ManOperationCm_typeAxis64PosInterface"(disableUnit := #disableUnit, SoftCamInterface := #AxisSoftCam[16], manualOperationEm := #manualOperationEm, manualOperationEmArea := #manualOperationEmArea[2], manualOperationCms := #manualOperationCms[16], Axis64Pos := #Axis64Pos[16], Status => #Status[16], errorID => #errorID[16])
   END_RUNG
   RUNG wire#powerrail
      { S7_Templates := "SrcType := Int" } LE_Contact(in1 := #tempUpperBoundAxis, in2 := 16)
      JumpCoil( TwoWayActuator )
   END_RUNG
   // the same network as SCL:
   "ManOperationCm_typeAxis64PosInterface"(disableUnit := #disableUnit,
                           SoftCamInterface := #AxisSoftCam[16],
                           manualOperationEm := #manualOperationEm,
                           manualOperationEmArea := #manualOperationEmArea[2],
                           manualOperationCms := #manualOperationCms[16],
                           Axis64Pos := #Axis64Pos[16],
                           Status => #Status[16],
                           errorID => #errorID[16]);
   IF #tempUpperBoundAxis <= 16 THEN GOTO TwoWayActuator; END_IF;
END_REGION

REGION Network 20: Equipment Module Area 2 Line 17
   RUNG wire#powerrail
      "ManOperationCm_typeAxis64PosInterface"(disableUnit := #disableUnit, SoftCamInterface := #AxisSoftCam[17], manualOperationEm := #manualOperationEm, manualOperationEmArea := #manualOperationEmArea[2], manualOperationCms := #manualOperationCms[17], Axis64Pos := #Axis64Pos[17], Status => #Status[17], errorID => #errorID[17])
   END_RUNG
   RUNG wire#powerrail
      { S7_Templates := "SrcType := Int" } LE_Contact(in1 := #tempUpperBoundAxis, in2 := 17)
      JumpCoil( TwoWayActuator )
   END_RUNG
   // the same network as SCL:
   "ManOperationCm_typeAxis64PosInterface"(disableUnit := #disableUnit,
                           SoftCamInterface := #AxisSoftCam[17],
                           manualOperationEm := #manualOperationEm,
                           manualOperationEmArea := #manualOperationEmArea[2],
                           manualOperationCms := #manualOperationCms[17],
                           Axis64Pos := #Axis64Pos[17],
                           Status => #Status[17],
                           errorID => #errorID[17]);
   IF #tempUpperBoundAxis <= 17 THEN GOTO TwoWayActuator; END_IF;
END_REGION

REGION Network 21: Equipment Module Area 2 Line 18
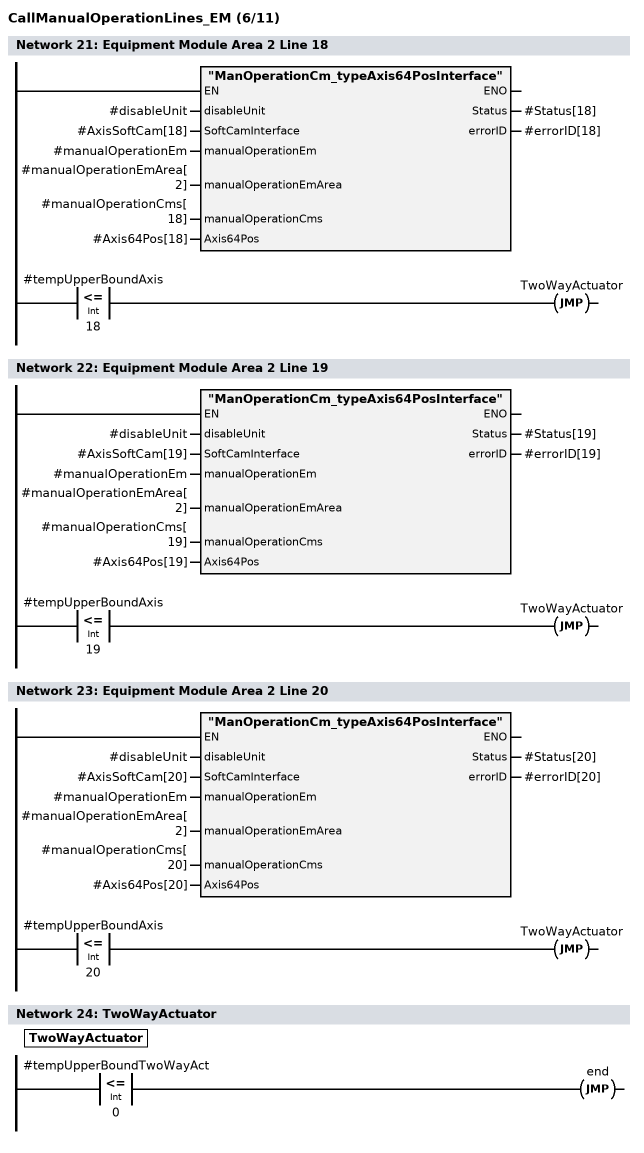
   RUNG wire#powerrail
      "ManOperationCm_typeAxis64PosInterface"(disableUnit := #disableUnit, SoftCamInterface := #AxisSoftCam[18], manualOperationEm := #manualOperationEm, manualOperationEmArea := #manualOperationEmArea[2], manualOperationCms := #manualOperationCms[18], Axis64Pos := #Axis64Pos[18], Status => #Status[18], errorID => #errorID[18])
   END_RUNG
   RUNG wire#powerrail
      { S7_Templates := "SrcType := Int" } LE_Contact(in1 := #tempUpperBoundAxis, in2 := 18)
      JumpCoil( TwoWayActuator )
   END_RUNG
   // the same network as SCL:
   "ManOperationCm_typeAxis64PosInterface"(disableUnit := #disableUnit,
                           SoftCamInterface := #AxisSoftCam[18],
                           manualOperationEm := #manualOperationEm,
                           manualOperationEmArea := #manualOperationEmArea[2],
                           manualOperationCms := #manualOperationCms[18],
                           Axis64Pos := #Axis64Pos[18],
                           Status => #Status[18],
                           errorID => #errorID[18]);
   IF #tempUpperBoundAxis <= 18 THEN GOTO TwoWayActuator; END_IF;
END_REGION

REGION Network 22: Equipment Module Area 2 Line 19
   RUNG wire#powerrail
      "ManOperationCm_typeAxis64PosInterface"(disableUnit := #disableUnit, SoftCamInterface := #AxisSoftCam[19], manualOperationEm := #manualOperationEm, manualOperationEmArea := #manualOperationEmArea[2], manualOperationCms := #manualOperationCms[19], Axis64Pos := #Axis64Pos[19], Status => #Status[19], errorID => #errorID[19])
   END_RUNG
   RUNG wire#powerrail
      { S7_Templates := "SrcType := Int" } LE_Contact(in1 := #tempUpperBoundAxis, in2 := 19)
      JumpCoil( TwoWayActuator )
   END_RUNG
   // the same network as SCL:
   "ManOperationCm_typeAxis64PosInterface"(disableUnit := #disableUnit,
                           SoftCamInterface := #AxisSoftCam[19],
                           manualOperationEm := #manualOperationEm,
                           manualOperationEmArea := #manualOperationEmArea[2],
                           manualOperationCms := #manualOperationCms[19],
                           Axis64Pos := #Axis64Pos[19],
                           Status => #Status[19],
                           errorID => #errorID[19]);
   IF #tempUpperBoundAxis <= 19 THEN GOTO TwoWayActuator; END_IF;
END_REGION

REGION Network 23: Equipment Module Area 2 Line 20
   RUNG wire#powerrail
      "ManOperationCm_typeAxis64PosInterface"(disableUnit := #disableUnit, SoftCamInterface := #AxisSoftCam[20], manualOperationEm := #manualOperationEm, manualOperationEmArea := #manualOperationEmArea[2], manualOperationCms := #manualOperationCms[20], Axis64Pos := #Axis64Pos[20], Status => #Status[20], errorID => #errorID[20])
   END_RUNG
   RUNG wire#powerrail
      { S7_Templates := "SrcType := Int" } LE_Contact(in1 := #tempUpperBoundAxis, in2 := 20)
      JumpCoil( TwoWayActuator )
   END_RUNG
   // the same network as SCL:
   "ManOperationCm_typeAxis64PosInterface"(disableUnit := #disableUnit,
                           SoftCamInterface := #AxisSoftCam[20],
                           manualOperationEm := #manualOperationEm,
                           manualOperationEmArea := #manualOperationEmArea[2],
                           manualOperationCms := #manualOperationCms[20],
                           Axis64Pos := #Axis64Pos[20],
                           Status => #Status[20],
                           errorID => #errorID[20]);
   IF #tempUpperBoundAxis <= 20 THEN GOTO TwoWayActuator; END_IF;
END_REGION

REGION Network 24: TwoWayActuator
   Label( TwoWayActuator )
   RUNG wire#powerrail
      { S7_Templates := "SrcType := Int" } LE_Contact(in1 := #tempUpperBoundTwoWayAct, in2 := 0)
      JumpCoil( end )
   END_RUNG
   // the same network as SCL:
   TwoWayActuator:
   IF #tempUpperBoundTwoWayAct <= 0 THEN GOTO end; END_IF;
END_REGION

REGION Network 25: Equipment Module Area 1 Line 21
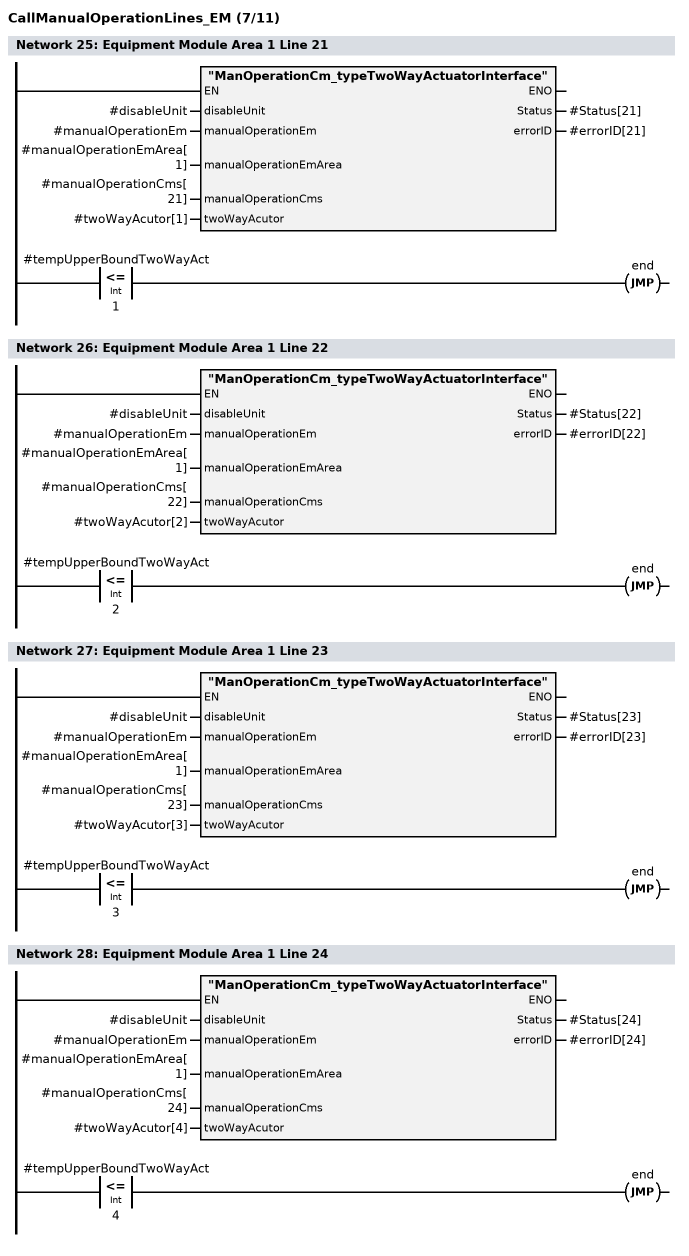
   RUNG wire#powerrail
      "ManOperationCm_typeTwoWayActuatorInterface"(disableUnit := #disableUnit, manualOperationEm := #manualOperationEm, manualOperationEmArea := #manualOperationEmArea[1], manualOperationCms := #manualOperationCms[21], twoWayAcutor := #twoWayAcutor[1], Status => #Status[21], errorID => #errorID[21])
   END_RUNG
   RUNG wire#powerrail
      { S7_Templates := "SrcType := Int" } LE_Contact(in1 := #tempUpperBoundTwoWayAct, in2 := 1)
      JumpCoil( end )
   END_RUNG
   // the same network as SCL:
   "ManOperationCm_typeTwoWayActuatorInterface"(disableUnit := #disableUnit,
                           manualOperationEm := #manualOperationEm,
                           manualOperationEmArea := #manualOperationEmArea[1],
                           manualOperationCms := #manualOperationCms[21],
                           twoWayAcutor := #twoWayAcutor[1],
                           Status => #Status[21],
                           errorID => #errorID[21]);
   IF #tempUpperBoundTwoWayAct <= 1 THEN GOTO end; END_IF;
END_REGION

REGION Network 26: Equipment Module Area 1 Line 22
   RUNG wire#powerrail
      "ManOperationCm_typeTwoWayActuatorInterface"(disableUnit := #disableUnit, manualOperationEm := #manualOperationEm, manualOperationEmArea := #manualOperationEmArea[1], manualOperationCms := #manualOperationCms[22], twoWayAcutor := #twoWayAcutor[2], Status => #Status[22], errorID => #errorID[22])
   END_RUNG
   RUNG wire#powerrail
      { S7_Templates := "SrcType := Int" } LE_Contact(in1 := #tempUpperBoundTwoWayAct, in2 := 2)
      JumpCoil( end )
   END_RUNG
   // the same network as SCL:
   "ManOperationCm_typeTwoWayActuatorInterface"(disableUnit := #disableUnit,
                           manualOperationEm := #manualOperationEm,
                           manualOperationEmArea := #manualOperationEmArea[1],
                           manualOperationCms := #manualOperationCms[22],
                           twoWayAcutor := #twoWayAcutor[2],
                           Status => #Status[22],
                           errorID => #errorID[22]);
   IF #tempUpperBoundTwoWayAct <= 2 THEN GOTO end; END_IF;
END_REGION

REGION Network 27: Equipment Module Area 1 Line 23
   RUNG wire#powerrail
      "ManOperationCm_typeTwoWayActuatorInterface"(disableUnit := #disableUnit, manualOperationEm := #manualOperationEm, manualOperationEmArea := #manualOperationEmArea[1], manualOperationCms := #manualOperationCms[23], twoWayAcutor := #twoWayAcutor[3], Status => #Status[23], errorID => #errorID[23])
   END_RUNG
   RUNG wire#powerrail
      { S7_Templates := "SrcType := Int" } LE_Contact(in1 := #tempUpperBoundTwoWayAct, in2 := 3)
      JumpCoil( end )
   END_RUNG
   // the same network as SCL:
   "ManOperationCm_typeTwoWayActuatorInterface"(disableUnit := #disableUnit,
                           manualOperationEm := #manualOperationEm,
                           manualOperationEmArea := #manualOperationEmArea[1],
                           manualOperationCms := #manualOperationCms[23],
                           twoWayAcutor := #twoWayAcutor[3],
                           Status => #Status[23],
                           errorID => #errorID[23]);
   IF #tempUpperBoundTwoWayAct <= 3 THEN GOTO end; END_IF;
END_REGION

REGION Network 28: Equipment Module Area 1 Line 24
   RUNG wire#powerrail
      "ManOperationCm_typeTwoWayActuatorInterface"(disableUnit := #disableUnit, manualOperationEm := #manualOperationEm, manualOperationEmArea := #manualOperationEmArea[1], manualOperationCms := #manualOperationCms[24], twoWayAcutor := #twoWayAcutor[4], Status => #Status[24], errorID => #errorID[24])
   END_RUNG
   RUNG wire#powerrail
      { S7_Templates := "SrcType := Int" } LE_Contact(in1 := #tempUpperBoundTwoWayAct, in2 := 4)
      JumpCoil( end )
   END_RUNG
   // the same network as SCL:
   "ManOperationCm_typeTwoWayActuatorInterface"(disableUnit := #disableUnit,
                           manualOperationEm := #manualOperationEm,
                           manualOperationEmArea := #manualOperationEmArea[1],
                           manualOperationCms := #manualOperationCms[24],
                           twoWayAcutor := #twoWayAcutor[4],
                           Status => #Status[24],
                           errorID => #errorID[24]);
   IF #tempUpperBoundTwoWayAct <= 4 THEN GOTO end; END_IF;
END_REGION

REGION Network 29: Equipment Module Area 1 Line 25
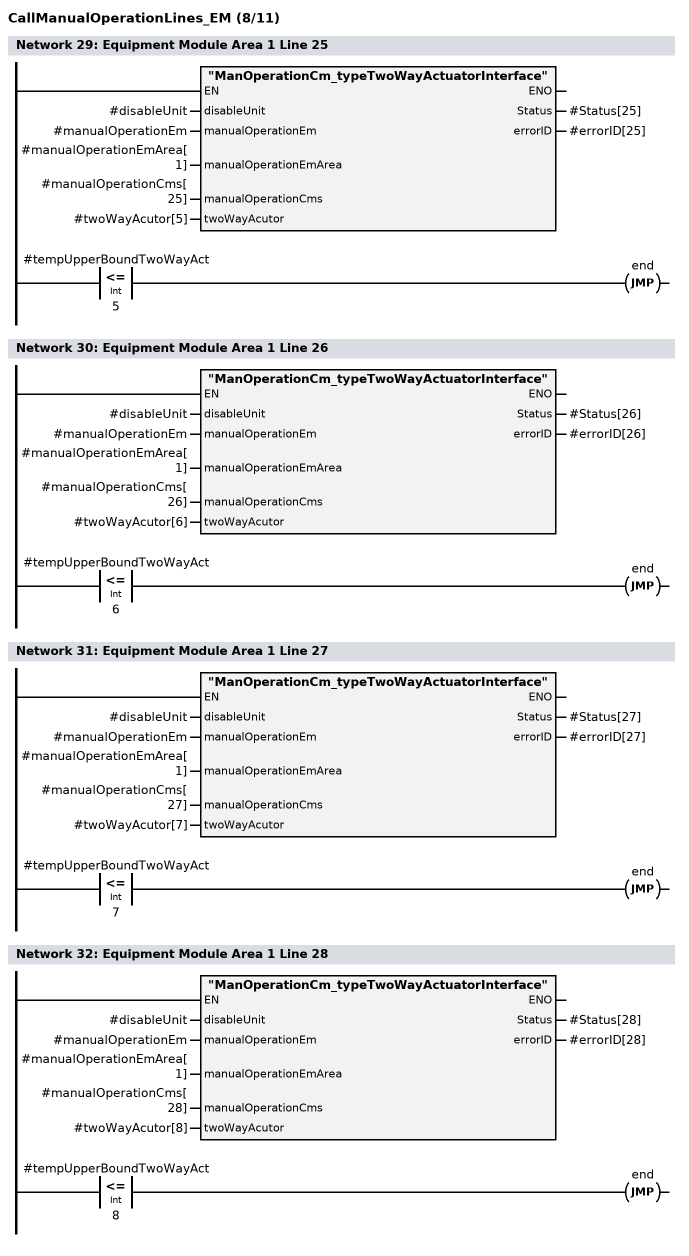
   RUNG wire#powerrail
      "ManOperationCm_typeTwoWayActuatorInterface"(disableUnit := #disableUnit, manualOperationEm := #manualOperationEm, manualOperationEmArea := #manualOperationEmArea[1], manualOperationCms := #manualOperationCms[25], twoWayAcutor := #twoWayAcutor[5], Status => #Status[25], errorID => #errorID[25])
   END_RUNG
   RUNG wire#powerrail
      { S7_Templates := "SrcType := Int" } LE_Contact(in1 := #tempUpperBoundTwoWayAct, in2 := 5)
      JumpCoil( end )
   END_RUNG
   // the same network as SCL:
   "ManOperationCm_typeTwoWayActuatorInterface"(disableUnit := #disableUnit,
                           manualOperationEm := #manualOperationEm,
                           manualOperationEmArea := #manualOperationEmArea[1],
                           manualOperationCms := #manualOperationCms[25],
                           twoWayAcutor := #twoWayAcutor[5],
                           Status => #Status[25],
                           errorID => #errorID[25]);
   IF #tempUpperBoundTwoWayAct <= 5 THEN GOTO end; END_IF;
END_REGION

REGION Network 30: Equipment Module Area 1 Line 26
   RUNG wire#powerrail
      "ManOperationCm_typeTwoWayActuatorInterface"(disableUnit := #disableUnit, manualOperationEm := #manualOperationEm, manualOperationEmArea := #manualOperationEmArea[1], manualOperationCms := #manualOperationCms[26], twoWayAcutor := #twoWayAcutor[6], Status => #Status[26], errorID => #errorID[26])
   END_RUNG
   RUNG wire#powerrail
      { S7_Templates := "SrcType := Int" } LE_Contact(in1 := #tempUpperBoundTwoWayAct, in2 := 6)
      JumpCoil( end )
   END_RUNG
   // the same network as SCL:
   "ManOperationCm_typeTwoWayActuatorInterface"(disableUnit := #disableUnit,
                           manualOperationEm := #manualOperationEm,
                           manualOperationEmArea := #manualOperationEmArea[1],
                           manualOperationCms := #manualOperationCms[26],
                           twoWayAcutor := #twoWayAcutor[6],
                           Status => #Status[26],
                           errorID => #errorID[26]);
   IF #tempUpperBoundTwoWayAct <= 6 THEN GOTO end; END_IF;
END_REGION

REGION Network 31: Equipment Module Area 1 Line 27
   RUNG wire#powerrail
      "ManOperationCm_typeTwoWayActuatorInterface"(disableUnit := #disableUnit, manualOperationEm := #manualOperationEm, manualOperationEmArea := #manualOperationEmArea[1], manualOperationCms := #manualOperationCms[27], twoWayAcutor := #twoWayAcutor[7], Status => #Status[27], errorID => #errorID[27])
   END_RUNG
   RUNG wire#powerrail
      { S7_Templates := "SrcType := Int" } LE_Contact(in1 := #tempUpperBoundTwoWayAct, in2 := 7)
      JumpCoil( end )
   END_RUNG
   // the same network as SCL:
   "ManOperationCm_typeTwoWayActuatorInterface"(disableUnit := #disableUnit,
                           manualOperationEm := #manualOperationEm,
                           manualOperationEmArea := #manualOperationEmArea[1],
                           manualOperationCms := #manualOperationCms[27],
                           twoWayAcutor := #twoWayAcutor[7],
                           Status => #Status[27],
                           errorID => #errorID[27]);
   IF #tempUpperBoundTwoWayAct <= 7 THEN GOTO end; END_IF;
END_REGION

REGION Network 32: Equipment Module Area 1 Line 28
   RUNG wire#powerrail
      "ManOperationCm_typeTwoWayActuatorInterface"(disableUnit := #disableUnit, manualOperationEm := #manualOperationEm, manualOperationEmArea := #manualOperationEmArea[1], manualOperationCms := #manualOperationCms[28], twoWayAcutor := #twoWayAcutor[8], Status => #Status[28], errorID => #errorID[28])
   END_RUNG
   RUNG wire#powerrail
      { S7_Templates := "SrcType := Int" } LE_Contact(in1 := #tempUpperBoundTwoWayAct, in2 := 8)
      JumpCoil( end )
   END_RUNG
   // the same network as SCL:
   "ManOperationCm_typeTwoWayActuatorInterface"(disableUnit := #disableUnit,
                           manualOperationEm := #manualOperationEm,
                           manualOperationEmArea := #manualOperationEmArea[1],
                           manualOperationCms := #manualOperationCms[28],
                           twoWayAcutor := #twoWayAcutor[8],
                           Status => #Status[28],
                           errorID => #errorID[28]);
   IF #tempUpperBoundTwoWayAct <= 8 THEN GOTO end; END_IF;
END_REGION

REGION Network 33: Equipment Module Area 1 Line 29
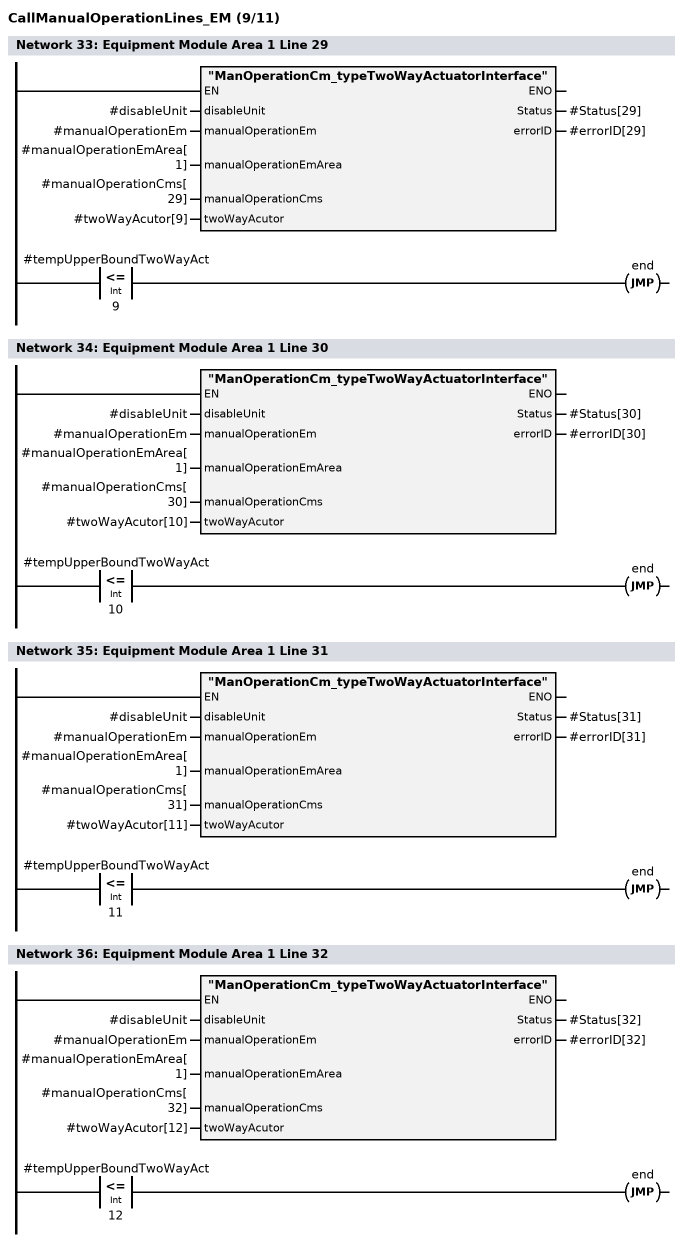
   RUNG wire#powerrail
      "ManOperationCm_typeTwoWayActuatorInterface"(disableUnit := #disableUnit, manualOperationEm := #manualOperationEm, manualOperationEmArea := #manualOperationEmArea[1], manualOperationCms := #manualOperationCms[29], twoWayAcutor := #twoWayAcutor[9], Status => #Status[29], errorID => #errorID[29])
   END_RUNG
   RUNG wire#powerrail
      { S7_Templates := "SrcType := Int" } LE_Contact(in1 := #tempUpperBoundTwoWayAct, in2 := 9)
      JumpCoil( end )
   END_RUNG
   // the same network as SCL:
   "ManOperationCm_typeTwoWayActuatorInterface"(disableUnit := #disableUnit,
                           manualOperationEm := #manualOperationEm,
                           manualOperationEmArea := #manualOperationEmArea[1],
                           manualOperationCms := #manualOperationCms[29],
                           twoWayAcutor := #twoWayAcutor[9],
                           Status => #Status[29],
                           errorID => #errorID[29]);
   IF #tempUpperBoundTwoWayAct <= 9 THEN GOTO end; END_IF;
END_REGION

REGION Network 34: Equipment Module Area 1 Line 30
   RUNG wire#powerrail
      "ManOperationCm_typeTwoWayActuatorInterface"(disableUnit := #disableUnit, manualOperationEm := #manualOperationEm, manualOperationEmArea := #manualOperationEmArea[1], manualOperationCms := #manualOperationCms[30], twoWayAcutor := #twoWayAcutor[10], Status => #Status[30], errorID => #errorID[30])
   END_RUNG
   RUNG wire#powerrail
      { S7_Templates := "SrcType := Int" } LE_Contact(in1 := #tempUpperBoundTwoWayAct, in2 := 10)
      JumpCoil( end )
   END_RUNG
   // the same network as SCL:
   "ManOperationCm_typeTwoWayActuatorInterface"(disableUnit := #disableUnit,
                           manualOperationEm := #manualOperationEm,
                           manualOperationEmArea := #manualOperationEmArea[1],
                           manualOperationCms := #manualOperationCms[30],
                           twoWayAcutor := #twoWayAcutor[10],
                           Status => #Status[30],
                           errorID => #errorID[30]);
   IF #tempUpperBoundTwoWayAct <= 10 THEN GOTO end; END_IF;
END_REGION

REGION Network 35: Equipment Module Area 1 Line 31
   RUNG wire#powerrail
      "ManOperationCm_typeTwoWayActuatorInterface"(disableUnit := #disableUnit, manualOperationEm := #manualOperationEm, manualOperationEmArea := #manualOperationEmArea[1], manualOperationCms := #manualOperationCms[31], twoWayAcutor := #twoWayAcutor[11], Status => #Status[31], errorID => #errorID[31])
   END_RUNG
   RUNG wire#powerrail
      { S7_Templates := "SrcType := Int" } LE_Contact(in1 := #tempUpperBoundTwoWayAct, in2 := 11)
      JumpCoil( end )
   END_RUNG
   // the same network as SCL:
   "ManOperationCm_typeTwoWayActuatorInterface"(disableUnit := #disableUnit,
                           manualOperationEm := #manualOperationEm,
                           manualOperationEmArea := #manualOperationEmArea[1],
                           manualOperationCms := #manualOperationCms[31],
                           twoWayAcutor := #twoWayAcutor[11],
                           Status => #Status[31],
                           errorID => #errorID[31]);
   IF #tempUpperBoundTwoWayAct <= 11 THEN GOTO end; END_IF;
END_REGION

REGION Network 36: Equipment Module Area 1 Line 32
   RUNG wire#powerrail
      "ManOperationCm_typeTwoWayActuatorInterface"(disableUnit := #disableUnit, manualOperationEm := #manualOperationEm, manualOperationEmArea := #manualOperationEmArea[1], manualOperationCms := #manualOperationCms[32], twoWayAcutor := #twoWayAcutor[12], Status => #Status[32], errorID => #errorID[32])
   END_RUNG
   RUNG wire#powerrail
      { S7_Templates := "SrcType := Int" } LE_Contact(in1 := #tempUpperBoundTwoWayAct, in2 := 12)
      JumpCoil( end )
   END_RUNG
   // the same network as SCL:
   "ManOperationCm_typeTwoWayActuatorInterface"(disableUnit := #disableUnit,
                           manualOperationEm := #manualOperationEm,
                           manualOperationEmArea := #manualOperationEmArea[1],
                           manualOperationCms := #manualOperationCms[32],
                           twoWayAcutor := #twoWayAcutor[12],
                           Status => #Status[32],
                           errorID => #errorID[32]);
   IF #tempUpperBoundTwoWayAct <= 12 THEN GOTO end; END_IF;
END_REGION

REGION Network 37: Equipment Module Area 1 Line 33
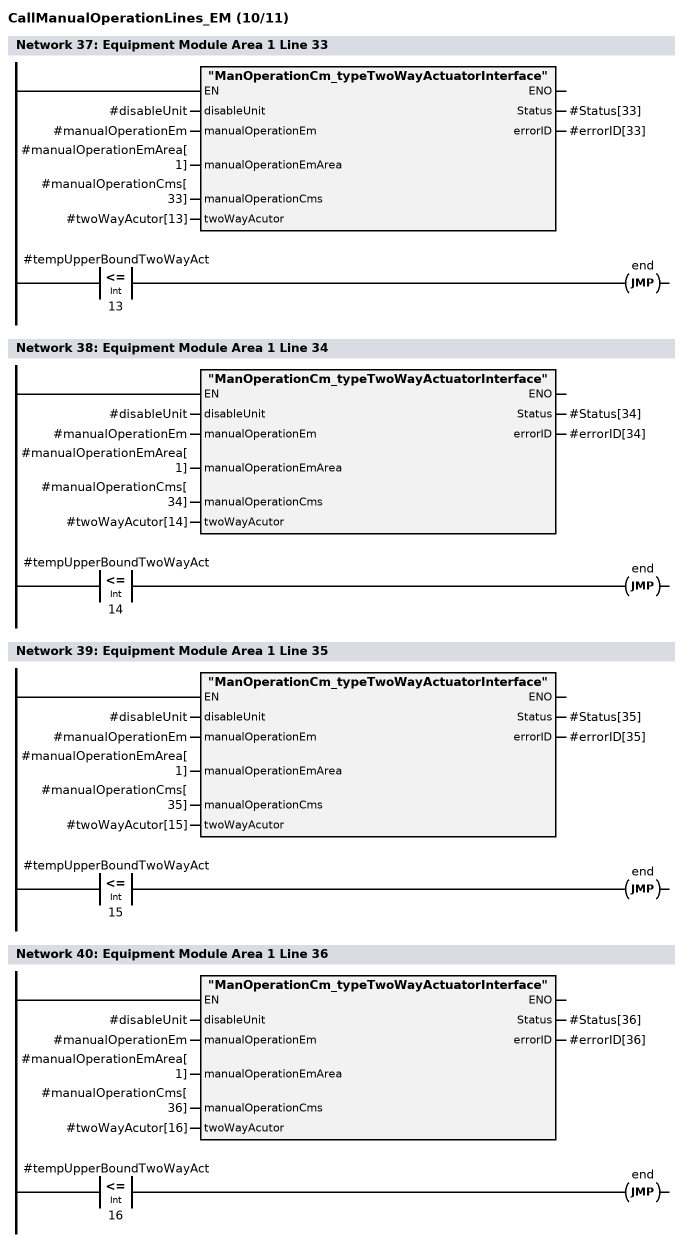
   RUNG wire#powerrail
      "ManOperationCm_typeTwoWayActuatorInterface"(disableUnit := #disableUnit, manualOperationEm := #manualOperationEm, manualOperationEmArea := #manualOperationEmArea[1], manualOperationCms := #manualOperationCms[33], twoWayAcutor := #twoWayAcutor[13], Status => #Status[33], errorID => #errorID[33])
   END_RUNG
   RUNG wire#powerrail
      { S7_Templates := "SrcType := Int" } LE_Contact(in1 := #tempUpperBoundTwoWayAct, in2 := 13)
      JumpCoil( end )
   END_RUNG
   // the same network as SCL:
   "ManOperationCm_typeTwoWayActuatorInterface"(disableUnit := #disableUnit,
                           manualOperationEm := #manualOperationEm,
                           manualOperationEmArea := #manualOperationEmArea[1],
                           manualOperationCms := #manualOperationCms[33],
                           twoWayAcutor := #twoWayAcutor[13],
                           Status => #Status[33],
                           errorID => #errorID[33]);
   IF #tempUpperBoundTwoWayAct <= 13 THEN GOTO end; END_IF;
END_REGION

REGION Network 38: Equipment Module Area 1 Line 34
   RUNG wire#powerrail
      "ManOperationCm_typeTwoWayActuatorInterface"(disableUnit := #disableUnit, manualOperationEm := #manualOperationEm, manualOperationEmArea := #manualOperationEmArea[1], manualOperationCms := #manualOperationCms[34], twoWayAcutor := #twoWayAcutor[14], Status => #Status[34], errorID => #errorID[34])
   END_RUNG
   RUNG wire#powerrail
      { S7_Templates := "SrcType := Int" } LE_Contact(in1 := #tempUpperBoundTwoWayAct, in2 := 14)
      JumpCoil( end )
   END_RUNG
   // the same network as SCL:
   "ManOperationCm_typeTwoWayActuatorInterface"(disableUnit := #disableUnit,
                           manualOperationEm := #manualOperationEm,
                           manualOperationEmArea := #manualOperationEmArea[1],
                           manualOperationCms := #manualOperationCms[34],
                           twoWayAcutor := #twoWayAcutor[14],
                           Status => #Status[34],
                           errorID => #errorID[34]);
   IF #tempUpperBoundTwoWayAct <= 14 THEN GOTO end; END_IF;
END_REGION

REGION Network 39: Equipment Module Area 1 Line 35
   RUNG wire#powerrail
      "ManOperationCm_typeTwoWayActuatorInterface"(disableUnit := #disableUnit, manualOperationEm := #manualOperationEm, manualOperationEmArea := #manualOperationEmArea[1], manualOperationCms := #manualOperationCms[35], twoWayAcutor := #twoWayAcutor[15], Status => #Status[35], errorID => #errorID[35])
   END_RUNG
   RUNG wire#powerrail
      { S7_Templates := "SrcType := Int" } LE_Contact(in1 := #tempUpperBoundTwoWayAct, in2 := 15)
      JumpCoil( end )
   END_RUNG
   // the same network as SCL:
   "ManOperationCm_typeTwoWayActuatorInterface"(disableUnit := #disableUnit,
                           manualOperationEm := #manualOperationEm,
                           manualOperationEmArea := #manualOperationEmArea[1],
                           manualOperationCms := #manualOperationCms[35],
                           twoWayAcutor := #twoWayAcutor[15],
                           Status => #Status[35],
                           errorID => #errorID[35]);
   IF #tempUpperBoundTwoWayAct <= 15 THEN GOTO end; END_IF;
END_REGION

REGION Network 40: Equipment Module Area 1 Line 36
   RUNG wire#powerrail
      "ManOperationCm_typeTwoWayActuatorInterface"(disableUnit := #disableUnit, manualOperationEm := #manualOperationEm, manualOperationEmArea := #manualOperationEmArea[1], manualOperationCms := #manualOperationCms[36], twoWayAcutor := #twoWayAcutor[16], Status => #Status[36], errorID => #errorID[36])
   END_RUNG
   RUNG wire#powerrail
      { S7_Templates := "SrcType := Int" } LE_Contact(in1 := #tempUpperBoundTwoWayAct, in2 := 16)
      JumpCoil( end )
   END_RUNG
   // the same network as SCL:
   "ManOperationCm_typeTwoWayActuatorInterface"(disableUnit := #disableUnit,
                           manualOperationEm := #manualOperationEm,
                           manualOperationEmArea := #manualOperationEmArea[1],
                           manualOperationCms := #manualOperationCms[36],
                           twoWayAcutor := #twoWayAcutor[16],
                           Status => #Status[36],
                           errorID => #errorID[36]);
   IF #tempUpperBoundTwoWayAct <= 16 THEN GOTO end; END_IF;
END_REGION

REGION Network 41: Equipment Module Area 1 Line 37
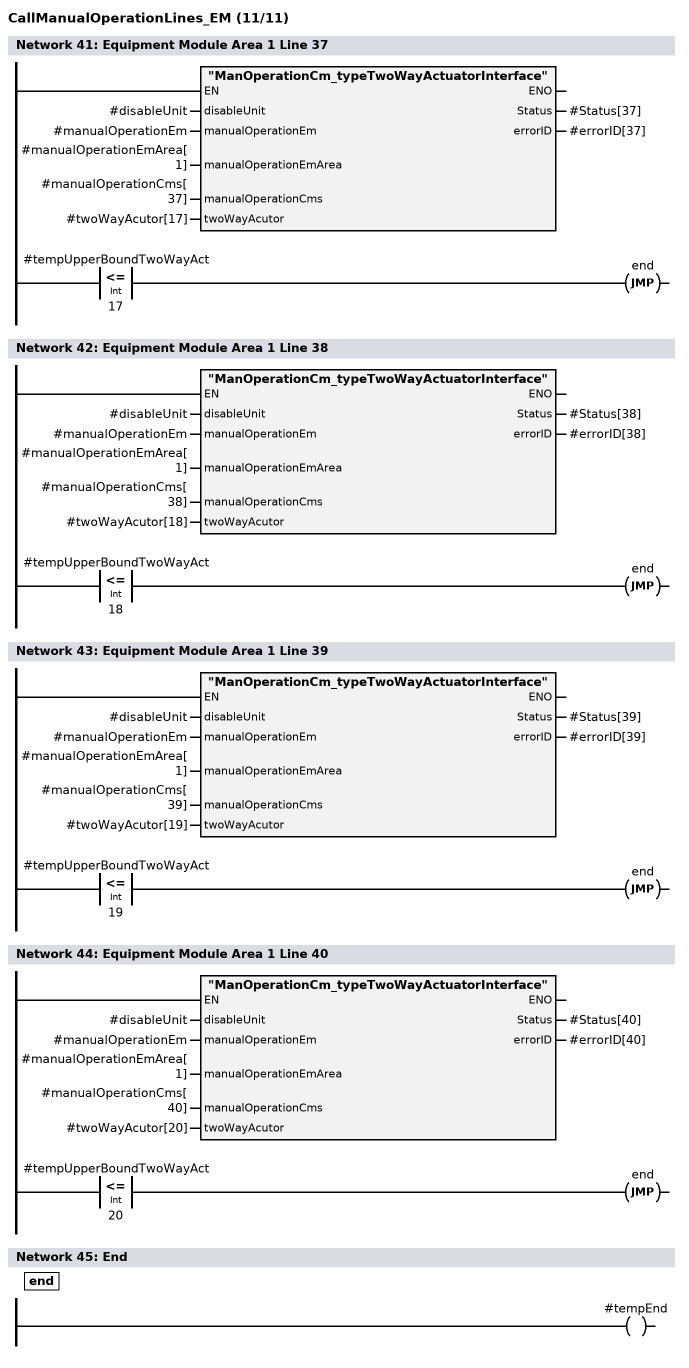
   RUNG wire#powerrail
      "ManOperationCm_typeTwoWayActuatorInterface"(disableUnit := #disableUnit, manualOperationEm := #manualOperationEm, manualOperationEmArea := #manualOperationEmArea[1], manualOperationCms := #manualOperationCms[37], twoWayAcutor := #twoWayAcutor[17], Status => #Status[37], errorID => #errorID[37])
   END_RUNG
   RUNG wire#powerrail
      { S7_Templates := "SrcType := Int" } LE_Contact(in1 := #tempUpperBoundTwoWayAct, in2 := 17)
      JumpCoil( end )
   END_RUNG
   // the same network as SCL:
   "ManOperationCm_typeTwoWayActuatorInterface"(disableUnit := #disableUnit,
                           manualOperationEm := #manualOperationEm,
                           manualOperationEmArea := #manualOperationEmArea[1],
                           manualOperationCms := #manualOperationCms[37],
                           twoWayAcutor := #twoWayAcutor[17],
                           Status => #Status[37],
                           errorID => #errorID[37]);
   IF #tempUpperBoundTwoWayAct <= 17 THEN GOTO end; END_IF;
END_REGION

REGION Network 42: Equipment Module Area 1 Line 38
   RUNG wire#powerrail
      "ManOperationCm_typeTwoWayActuatorInterface"(disableUnit := #disableUnit, manualOperationEm := #manualOperationEm, manualOperationEmArea := #manualOperationEmArea[1], manualOperationCms := #manualOperationCms[38], twoWayAcutor := #twoWayAcutor[18], Status => #Status[38], errorID => #errorID[38])
   END_RUNG
   RUNG wire#powerrail
      { S7_Templates := "SrcType := Int" } LE_Contact(in1 := #tempUpperBoundTwoWayAct, in2 := 18)
      JumpCoil( end )
   END_RUNG
   // the same network as SCL:
   "ManOperationCm_typeTwoWayActuatorInterface"(disableUnit := #disableUnit,
                           manualOperationEm := #manualOperationEm,
                           manualOperationEmArea := #manualOperationEmArea[1],
                           manualOperationCms := #manualOperationCms[38],
                           twoWayAcutor := #twoWayAcutor[18],
                           Status => #Status[38],
                           errorID => #errorID[38]);
   IF #tempUpperBoundTwoWayAct <= 18 THEN GOTO end; END_IF;
END_REGION

REGION Network 43: Equipment Module Area 1 Line 39
   RUNG wire#powerrail
      "ManOperationCm_typeTwoWayActuatorInterface"(disableUnit := #disableUnit, manualOperationEm := #manualOperationEm, manualOperationEmArea := #manualOperationEmArea[1], manualOperationCms := #manualOperationCms[39], twoWayAcutor := #twoWayAcutor[19], Status => #Status[39], errorID => #errorID[39])
   END_RUNG
   RUNG wire#powerrail
      { S7_Templates := "SrcType := Int" } LE_Contact(in1 := #tempUpperBoundTwoWayAct, in2 := 19)
      JumpCoil( end )
   END_RUNG
   // the same network as SCL:
   "ManOperationCm_typeTwoWayActuatorInterface"(disableUnit := #disableUnit,
                           manualOperationEm := #manualOperationEm,
                           manualOperationEmArea := #manualOperationEmArea[1],
                           manualOperationCms := #manualOperationCms[39],
                           twoWayAcutor := #twoWayAcutor[19],
                           Status => #Status[39],
                           errorID => #errorID[39]);
   IF #tempUpperBoundTwoWayAct <= 19 THEN GOTO end; END_IF;
END_REGION

REGION Network 44: Equipment Module Area 1 Line 40
   RUNG wire#powerrail
      "ManOperationCm_typeTwoWayActuatorInterface"(disableUnit := #disableUnit, manualOperationEm := #manualOperationEm, manualOperationEmArea := #manualOperationEmArea[1], manualOperationCms := #manualOperationCms[40], twoWayAcutor := #twoWayAcutor[20], Status => #Status[40], errorID => #errorID[40])
   END_RUNG
   RUNG wire#powerrail
      { S7_Templates := "SrcType := Int" } LE_Contact(in1 := #tempUpperBoundTwoWayAct, in2 := 20)
      JumpCoil( end )
   END_RUNG
   // the same network as SCL:
   "ManOperationCm_typeTwoWayActuatorInterface"(disableUnit := #disableUnit,
                           manualOperationEm := #manualOperationEm,
                           manualOperationEmArea := #manualOperationEmArea[1],
                           manualOperationCms := #manualOperationCms[40],
                           twoWayAcutor := #twoWayAcutor[20],
                           Status => #Status[40],
                           errorID => #errorID[40]);
   IF #tempUpperBoundTwoWayAct <= 20 THEN GOTO end; END_IF;
END_REGION

REGION Network 45: End
   Label( end )
   RUNG wire#powerrail
      Coil( #tempEnd )
   END_RUNG
   // the same network as SCL:
   end:
   #tempEnd := TRUE;
END_REGION
END_FUNCTION

FUNCTION "ManOperationCm_typeAxis64PosInterface" : Void   // FC74, LAD
// stored: SetENOAutomatically false
   VAR_INPUT
      disableUnit : Bool;
      SoftCamInterface : "LER_typeSoftCamRelation";
   END_VAR
   VAR_OUTPUT
      Status : Word;
      errorID : Word;
   END_VAR
   VAR_IN_OUT
      manualOperationEm : "LAF_typeManEm";
      manualOperationEmArea : "LAF_typeManOperationArea";
      manualOperationCms : "LAF_typeManOperation";
      Axis64Pos : "LBC_typeAxis64PosInterface";
   END_VAR
   VAR_TEMP
      tempMaxPos : LReal;
      tempIndex : Int;
   END_VAR
BEGIN

REGION Network 1 (SCL): MaxPos Find
   FOR #tempIndex := 0 TO 15 DO
       IF #Axis64Pos.configuration.setPositions[#tempIndex].position > #tempMaxPos THEN
           #tempMaxPos := #Axis64Pos.configuration.setPositions[#tempIndex].position;
       END_IF;
   END_FOR;
END_REGION

